LIN {X 0,Y 362.111,Z 381.376,A -85,B 0,C 180,E1 -12954.431,E2 -12954.431} C_VEL
LIN {X 0,Y 362.275,Z 381.356,A -85,B 0,C 180,E1 -12957.776,E2 -12957.776} C_VEL
LIN {X 0,Y 362.422,Z 381.337,A -85,B 0,C 180,E1 -12960,E2 -12960} C_VEL
LIN {X 0,Y 362.276,Z 381.354,A -85,B 0,C 180,E1 -12962.224,E2 -12962.224} C_VEL
LIN {X 0,Y 362.165,Z 381.372,A -85,B 0,C 180,E1 -12966.686,E2 -12966.686} C_VEL
LIN {X 0,Y 362.068,Z 381.386,A -85,B 0,C 180,E1 -12968.933,E2 -12968.933} C_VEL
LIN {X 0,Y 361.959,Z 381.395,A -85,B 0,C 180,E1 -12972.332,E2 -12972.332} C_VEL
LIN {X 0,Y 361.955,Z 381.398,A -85,B 0,C 180,E1 -12974.621,E2 -12974.621} C_VEL
LIN {X 0,Y 361.949,Z 381.396,A -85,B 0,C 180,E1 -12978.1,E2 -12978.1} C_VEL
LIN {X 0,Y 361.885,Z 381.404,A -85,B 0,C 180,E1 -12981.653,E2 -12981.653} C_VEL
LIN {X 0,Y 361.922,Z 381.4,A -85,B 0,C 180,E1 -12985.291,E2 -12985.291} C_VEL
LIN {X 0,Y 361.912,Z 381.4,A -85,B 0,C 180,E1 -12987.779,E2 -12987.779} C_VEL
LIN {X 0,Y 361.841,Z 381.41,A -85,B 0,C 180,E1 -12991.286,E2 -12991.286} C_VEL
LIN {X 0,Y 361.849,Z 381.411,A -85,B 0,C 180,E1 -12994.281,E2 -12994.281} C_VEL
LIN {X 0,Y 361.861,Z 381.407,A -85,B 0,C 180,E1 -12997.224,E2 -12997.224} C_VEL
LIN {X 0,Y 361.901,Z 381.405,A -85,B 0,C 180,E1 -13000.769,E2 -13000.769} C_VEL
LIN {X 0,Y 361.907,Z 381.406,A -85,B 0,C 180,E1 -13004.355,E2 -13004.355} C_VEL
LIN {X 0,Y 361.838,Z 381.41,A -85,B 0,C 180,E1 -13007.568,E2 -13007.568} C_VEL
LIN {X 0,Y 361.87,Z 381.407,A -85,B 0,C 180,E1 -13010.974,E2 -13010.974} C_VEL
LIN {X 0,Y 361.873,Z 381.408,A -85,B 0,C 180,E1 -13014.656,E2 -13014.656} C_VEL
LIN {X 0,Y 361.837,Z 381.416,A -85,B 0,C 180,E1 -13018.371,E2 -13018.371} C_VEL
LIN {X 0,Y 361.92,Z 381.554,A -85,B 0,C 180,E1 -13019.486,E2 -13019.486} C_VEL
LIN {X 0,Y 364.634,Z 393.775,A -85,B 0,C 180,E1 -13022.697,E2 -13022.697} C_VEL
LIN {X 0,Y 366.023,Z 401.747,A -85,B 0,C 180,E1 -13024.694,E2 -13024.694} C_VEL
LIN {X 0,Y 364.596,Z 415.783,A -85,B 0,C 180,E1 -13027.91,E2 -13027.91} C_VEL
LIN {X 0,Y 369.128,Z 442.935,A -85,B 0,C 180,E1 -13028.748,E2 -13028.748} C_VEL
LIN {X 0,Y 370.192,Z 451.075,A -85,B 0,C 180,E1 -13028.977,E2 -13028.977} C_VEL
LIN {X 0,Y 368.952,Z 524.302,A -85,B 0,C 180,E1 -13030.42,E2 -13030.42} C_VEL
LIN {X 0,Y 368.284,Z 537.515,A -85,B 0,C 180,E1 -13030.89,E2 -13030.89} C_VEL
LIN {X 0,Y 367.403,Z 549.648,A -85,B 0,C 180,E1 -13031.53,E2 -13031.53} C_VEL
LIN {X 0,Y 366.36,Z 561.898,A -85,B 0,C 180,E1 -13032.414,E2 -13032.414} C_VEL
LIN {X 0,Y 365.162,Z 573.49,A -85,B 0,C 180,E1 -13033.508,E2 -13033.508} C_VEL
LIN {X 0,Y 364.028,Z 584.075,A -85,B 0,C 180,E1 -13034.768,E2 -13034.768} C_VEL
LIN {X 0,Y 363.201,Z 592.48,A -85,B 0,C 180,E1 -13036.003,E2 -13036.003} C_VEL
LIN {X 0,Y 362.381,Z 600.367,A -85,B 0,C 180,E1 -13037.398,E2 -13037.398} C_VEL
LIN {X 0,Y 361.507,Z 608.07,A -85,B 0,C 180,E1 -13039.074,E2 -13039.074} C_VEL
LIN {X 0,Y 360.907,Z 615.183,A -85,B 0,C 180,E1 -13041.038,E2 -13041.038} C_VEL
LIN {X 0,Y 360.587,Z 619.917,A -85,B 0,C 180,E1 -13042.722,E2 -13042.722} C_VEL
LIN {X 0,Y 360.383,Z 623.535,A -85,B 0,C 180,E1 -13044.404,E2 -13044.404} C_VEL
LIN {X 0,Y 360.365,Z 625.404,A -85,B 0,C 180,E1 -13045.526,E2 -13045.526} C_VEL
LIN {X 0,Y 360.303,Z 626.804,A -85,B 0,C 180,E1 -13046.645,E2 -13046.645} C_VEL
LIN {X 0,Y 360.385,Z 628.417,A -85,B 0,C 180,E1 -13048.883,E2 -13048.883} C_VEL
LIN {X 0,Y 360.424,Z 628.634,A -85,B 0,C 180,E1 -13050,E2 -13050} C_VEL
LIN {X 0,Y 360.385,Z 628.413,A -85,B 0,C 180,E1 -13051.117,E2 -13051.117} C_VEL
LIN {X 0,Y 360.304,Z 626.796,A -85,B 0,C 180,E1 -13053.355,E2 -13053.355} C_VEL
LIN {X 0,Y 360.366,Z 625.392,A -85,B 0,C 180,E1 -13054.474,E2 -13054.474} C_VEL
LIN {X 0,Y 360.378,Z 622.815,A -85,B 0,C 180,E1 -13055.961,E2 -13055.961} C_VEL
LIN {X 0,Y 360.66,Z 618.449,A -85,B 0,C 180,E1 -13057.84,E2 -13057.84} C_VEL
LIN {X 0,Y 361.127,Z 612.315,A -85,B 0,C 180,E1 -13059.804,E2 -13059.804} C_VEL
LIN {X 0,Y 361.753,Z 605.619,A -85,B 0,C 180,E1 -13061.486,E2 -13061.486} C_VEL
LIN {X 0,Y 362.739,Z 597.321,A -85,B 0,C 180,E1 -13063.159,E2 -13063.159} C_VEL
LIN {X 0,Y 363.749,Z 587.774,A -85,B 0,C 180,E1 -13064.699,E2 -13064.699} C_VEL
LIN {X 0,Y 364.751,Z 577.122,A -85,B 0,C 180,E1 -13066.079,E2 -13066.079} C_VEL
LIN {X 0,Y 365.892,Z 566.481,A -85,B 0,C 180,E1 -13067.176,E2 -13067.176} C_VEL
LIN {X 0,Y 366.968,Z 554.588,A -85,B 0,C 180,E1 -13068.132,E2 -13068.132} C_VEL
LIN {X 0,Y 367.917,Z 542.215,A -85,B 0,C 180,E1 -13068.877,E2 -13068.877} C_VEL
LIN {X 0,Y 368.713,Z 529.503,A -85,B 0,C 180,E1 -13069.412,E2 -13069.412} C_VEL
LIN {X 0,Y 369.102,Z 516.14,A -85,B 0,C 180,E1 -13069.753,E2 -13069.753} C_VEL
LIN {X 0,Y 370.066,Z 449.66,A -85,B 0,C 180,E1 -13071.046,E2 -13071.046} C_VEL
LIN {X 0,Y 365.283,Z 419.717,A -85,B 0,C 180,E1 -13071.95,E2 -13071.95} C_VEL
LIN {X 0,Y 364.608,Z 415.73,A -85,B 0,C 180,E1 -13072.09,E2 -13072.09} C_VEL
LIN {X 0,Y 366.013,Z 401.695,A -85,B 0,C 180,E1 -13075.303,E2 -13075.303} C_VEL
LIN {X 0,Y 363.854,Z 390.071,A -85,B 0,C 180,E1 -13078.243,E2 -13078.243} C_VEL
LIN {X 0,Y 361.9,Z 381.408,A -85,B 0,C 180,E1 -13080.554,E2 -13080.554} C_VEL
LIN {X 0,Y 361.853,Z 381.409,A -85,B 0,C 180,E1 -13084.28,E2 -13084.28} C_VEL
LIN {X 0,Y 361.869,Z 381.408,A -85,B 0,C 180,E1 -13087.224,E2 -13087.224} C_VEL
LIN {X 0,Y 361.852,Z 381.408,A -85,B 0,C 180,E1 -13090.758,E2 -13090.758} C_VEL
LIN {X 0,Y 361.844,Z 381.409,A -85,B 0,C 180,E1 -13094.363,E2 -13094.363} C_VEL
LIN {X 0,Y 361.88,Z 381.41,A -85,B 0,C 180,E1 -13097.559,E2 -13097.559} C_VEL
LIN {X 0,Y 361.871,Z 381.407,A -85,B 0,C 180,E1 -13100.972,E2 -13100.972} C_VEL
LIN {X 0,Y 361.869,Z 381.406,A -85,B 0,C 180,E1 -13104.654,E2 -13104.654} C_VEL
LIN {X 0,Y 361.832,Z 381.41,A -85,B 0,C 180,E1 -13108.37,E2 -13108.37} C_VEL
LIN {X 0,Y 361.896,Z 381.405,A -85,B 0,C 180,E1 -13110.955,E2 -13110.955} C_VEL
LIN {X 0,Y 361.948,Z 381.4,A -85,B 0,C 180,E1 -13113.475,E2 -13113.475} C_VEL
LIN {X 0,Y 361.884,Z 381.409,A -85,B 0,C 180,E1 -13117.144,E2 -13117.144} C_VEL
LIN {X 0,Y 361.899,Z 381.403,A -85,B 0,C 180,E1 -13120.723,E2 -13120.723} C_VEL
LIN {X 0,Y 361.926,Z 381.403,A -85,B 0,C 180,E1 -13123.066,E2 -13123.066} C_VEL
LIN {X 0,Y 361.993,Z 381.391,A -85,B 0,C 180,E1 -13126.528,E2 -13126.528} C_VEL
LIN {X 0,Y 362.029,Z 381.385,A -85,B 0,C 180,E1 -13129.938,E2 -13129.938} C_VEL
LIN {X 0,Y 362.143,Z 381.371,A -85,B 0,C 180,E1 -13132.192,E2 -13132.192} C_VEL
LIN {X 0,Y 362.111,Z 381.376,A -85,B 0,C 180,E1 -13134.431,E2 -13134.431} C_VEL
LIN {X 0,Y 362.276,Z 381.355,A -85,B 0,C 180,E1 -13137.776,E2 -13137.776} C_VEL
LIN {X 0,Y 362.422,Z 381.337,A -85,B 0,C 180,E1 -13140,E2 -13140} C_VEL
LIN {X 0,Y 362.276,Z 381.355,A -85,B 0,C 180,E1 -13142.224,E2 -13142.224} C_VEL
LIN {X 0,Y 362.165,Z 381.373,A -85,B 0,C 180,E1 -13146.686,E2 -13146.686} C_VEL
LIN {X 0,Y 362.068,Z 381.386,A -85,B 0,C 180,E1 -13148.933,E2 -13148.933} C_VEL
LIN {X 0,Y 361.959,Z 381.396,A -85,B 0,C 180,E1 -13152.332,E2 -13152.332} C_VEL
LIN {X 0,Y 361.955,Z 381.4,A -85,B 0,C 180,E1 -13154.621,E2 -13154.621} C_VEL
LIN {X 0,Y 361.953,Z 381.396,A -85,B 0,C 180,E1 -13158.1,E2 -13158.1} C_VEL
LIN {X 0,Y 361.886,Z 381.403,A -85,B 0,C 180,E1 -13161.653,E2 -13161.653} C_VEL
LIN {X 0,Y 361.922,Z 381.399,A -85,B 0,C 180,E1 -13165.291,E2 -13165.291} C_VEL
LIN {X 0,Y 361.912,Z 381.4,A -85,B 0,C 180,E1 -13167.779,E2 -13167.779} C_VEL
LIN {X 0,Y 361.841,Z 381.409,A -85,B 0,C 180,E1 -13171.286,E2 -13171.286} C_VEL
LIN {X 0,Y 361.849,Z 381.412,A -85,B 0,C 180,E1 -13174.281,E2 -13174.281} C_VEL
LIN {X 0,Y 361.861,Z 381.407,A -85,B 0,C 180,E1 -13177.224,E2 -13177.224} C_VEL
LIN {X 0,Y 361.902,Z 381.404,A -85,B 0,C 180,E1 -13180.769,E2 -13180.769} C_VEL
LIN {X 0,Y 361.9,Z 381.408,A -85,B 0,C 180,E1 -13184.356,E2 -13184.356} C_VEL
LIN {X 0,Y 361.835,Z 381.41,A -85,B 0,C 180,E1 -13187.569,E2 -13187.569} C_VEL
LIN {X 0,Y 361.87,Z 381.406,A -85,B 0,C 180,E1 -13191.577,E2 -13191.577} C_VEL
LIN {X 0,Y 361.873,Z 381.407,A -85,B 0,C 180,E1 -13194.656,E2 -13194.656} C_VEL
LIN {X 0,Y 361.837,Z 381.414,A -85,B 0,C 180,E1 -13198.371,E2 -13198.371} C_VEL
LIN {X 0,Y 361.909,Z 381.405,A -85,B 0,C 180,E1 -13202.222,E2 -13202.222} C_VEL
LIN {X 0,Y 361.931,Z 381.511,A -85,B 0,C 180,E1 -13205,E2 -13205} C_VEL
LIN {X 0,Y 363.858,Z 391.181,A -85,B 0,C 180,E1 -13207.922,E2 -13207.922} C_VEL
LIN {X 0,Y 367.858,Z 402.665,A -85,B 0,C 180,E1 -13208.433,E2 -13208.433} C_VEL
LIN {X 0,Y 370.625,Z 416.292,A -85,B 0,C 180,E1 -13208.883,E2 -13208.883} C_VEL
LIN {X 0,Y 369.277,Z 498.572,A -85,B 0,C 180,E1 -13210.51,E2 -13210.51} C_VEL
LIN {X 0,Y 368.645,Z 512.357,A -85,B 0,C 180,E1 -13211.018,E2 -13211.018} C_VEL
LIN {X 0,Y 367.922,Z 524.708,A -85,B 0,C 180,E1 -13211.701,E2 -13211.701} C_VEL
LIN {X 0,Y 367.034,Z 536.529,A -85,B 0,C 180,E1 -13212.592,E2 -13212.592} C_VEL
LIN {X 0,Y 366.058,Z 547.685,A -85,B 0,C 180,E1 -13213.673,E2 -13213.673} C_VEL
LIN {X 0,Y 365.101,Z 558.085,A -85,B 0,C 180,E1 -13214.938,E2 -13214.938} C_VEL
LIN {X 0,Y 364.055,Z 567.253,A -85,B 0,C 180,E1 -13216.321,E2 -13216.321} C_VEL
LIN {X 0,Y 362.98,Z 576.155,A -85,B 0,C 180,E1 -13217.987,E2 -13217.987} C_VEL
LIN {X 0,Y 362.153,Z 583.316,A -85,B 0,C 180,E1 -13219.659,E2 -13219.659} C_VEL
LIN {X 0,Y 361.582,Z 588.146,A -85,B 0,C 180,E1 -13221.055,E2 -13221.055} C_VEL
LIN {X 0,Y 361.087,Z 592.838,A -85,B 0,C 180,E1 -13222.733,E2 -13222.733} C_VEL
LIN {X 0,Y 360.833,Z 596.422,A -85,B 0,C 180,E1 -13224.411,E2 -13224.411} C_VEL
LIN {X 0,Y 360.604,Z 598.279,A -85,B 0,C 180,E1 -13225.529,E2 -13225.529} C_VEL
LIN {X 0,Y 360.497,Z 599.674,A -85,B 0,C 180,E1 -13226.647,E2 -13226.647} C_VEL
LIN {X 0,Y 360.421,Z 601.275,A -85,B 0,C 180,E1 -13228.883,E2 -13228.883} C_VEL
LIN {X 0,Y 360.426,Z 601.507,A -85,B 0,C 180,E1 -13230,E2 -13230} C_VEL
LIN {X 0,Y 360.421,Z 601.318,A -85,B 0,C 180,E1 -13231.117,E2 -13231.117} C_VEL
LIN {X 0,Y 360.456,Z 600.735,A -85,B 0,C 180,E1 -13232.235,E2 -13232.235} C_VEL
LIN {X 0,Y 360.602,Z 598.419,A -85,B 0,C 180,E1 -13234.471,E2 -13234.471} C_VEL
LIN {X 0,Y 360.93,Z 595.557,A -85,B 0,C 180,E1 -13236.148,E2 -13236.148} C_VEL
LIN {X 0,Y 361.226,Z 591.682,A -85,B 0,C 180,E1 -13237.827,E2 -13237.827} C_VEL
LIN {X 0,Y 361.741,Z 586.677,A -85,B 0,C 180,E1 -13239.505,E2 -13239.505} C_VEL
LIN {X 0,Y 362.473,Z 580.373,A -85,B 0,C 180,E1 -13241.18,E2 -13241.18} C_VEL
LIN {X 0,Y 363.389,Z 572.48,A -85,B 0,C 180,E1 -13242.85,E2 -13242.85} C_VEL
LIN {X 0,Y 364.398,Z 564.427,A -85,B 0,C 180,E1 -13244.235,E2 -13244.235} C_VEL
LIN {X 0,Y 365.437,Z 554.603,A -85,B 0,C 180,E1 -13245.619,E2 -13245.619} C_VEL
LIN {X 0,Y 366.306,Z 544.935,A -85,B 0,C 180,E1 -13246.725,E2 -13246.725} C_VEL
LIN {X 0,Y 367.254,Z 534.463,A -85,B 0,C 180,E1 -13247.685,E2 -13247.685} C_VEL
LIN {X 0,Y 368.214,Z 521.847,A -85,B 0,C 180,E1 -13248.572,E2 -13248.572} C_VEL
LIN {X 0,Y 368.838,Z 509.216,A -85,B 0,C 180,E1 -13249.225,E2 -13249.225} C_VEL
LIN {X 0,Y 369.326,Z 497.213,A -85,B 0,C 180,E1 -13249.632,E2 -13249.632} C_VEL
LIN {X 0,Y 369.596,Z 480.297,A -85,B 0,C 180,E1 -13249.98,E2 -13249.98} C_VEL
LIN {X 0,Y 369.082,Z 474.486,A -85,B 0,C 180,E1 -13250.127,E2 -13250.127} C_VEL
LIN {X 0,Y 364.083,Z 455.777,A -85,B 0,C 180,E1 -13250.807,E2 -13250.807} C_VEL
LIN {X 0,Y 363.551,Z 449.967,A -85,B 0,C 180,E1 -13250.959,E2 -13250.959} C_VEL
LIN {X 0,Y 363.969,Z 416.729,A -85,B 0,C 180,E1 -13251.624,E2 -13251.624} C_VEL
LIN {X 0,Y 360.737,Z 402.305,A -85,B 0,C 180,E1 -13252.134,E2 -13252.134} C_VEL
LIN {X 0,Y 356.684,Z 391.491,A -85,B 0,C 180,E1 -13252.648,E2 -13252.648} C_VEL
LIN {X 0,Y 354.901,Z 382.279,A -85,B 0,C 180,E1 -13255.512,E2 -13255.512} C_VEL
LIN {X 0,Y 354.846,Z 382.283,A -85,B 0,C 180,E1 -13258.381,E2 -13258.381} C_VEL
LIN {X 0,Y 354.787,Z 382.29,A -85,B 0,C 180,E1 -13262.333,E2 -13262.333} C_VEL
LIN {X 0,Y 354.821,Z 382.288,A -85,B 0,C 180,E1 -13265.699,E2 -13265.699} C_VEL
LIN {X 0,Y 354.822,Z 382.286,A -85,B 0,C 180,E1 -13269.423,E2 -13269.423} C_VEL
LIN {X 0,Y 354.788,Z 382.287,A -85,B 0,C 180,E1 -13272.867,E2 -13272.867} C_VEL
LIN {X 0,Y 354.837,Z 382.283,A -85,B 0,C 180,E1 -13276.114,E2 -13276.114} C_VEL
LIN {X 0,Y 354.854,Z 382.28,A -85,B 0,C 180,E1 -13279.188,E2 -13279.188} C_VEL
LIN {X 0,Y 354.805,Z 382.285,A -85,B 0,C 180,E1 -13282.401,E2 -13282.401} C_VEL
LIN {X 0,Y 354.808,Z 382.286,A -85,B 0,C 180,E1 -13284.94,E2 -13284.94} C_VEL
LIN {X 0,Y 354.789,Z 382.288,A -85,B 0,C 180,E1 -13288.404,E2 -13288.404} C_VEL
LIN {X 0,Y 354.845,Z 382.285,A -85,B 0,C 180,E1 -13291.618,E2 -13291.618} C_VEL
LIN {X 0,Y 354.893,Z 382.275,A -85,B 0,C 180,E1 -13294.172,E2 -13294.172} C_VEL
LIN {X 0,Y 354.829,Z 382.284,A -85,B 0,C 180,E1 -13297.893,E2 -13297.893} C_VEL
LIN {X 0,Y 354.916,Z 382.272,A -85,B 0,C 180,E1 -13301.891,E2 -13301.891} C_VEL
LIN {X 0,Y 354.936,Z 382.27,A -85,B 0,C 180,E1 -13305.981,E2 -13305.981} C_VEL
LIN {X 0,Y 354.975,Z 382.266,A -85,B 0,C 180,E1 -13309.736,E2 -13309.736} C_VEL
LIN {X 0,Y 355.106,Z 382.248,A -85,B 0,C 180,E1 -13312.037,E2 -13312.037} C_VEL
LIN {X 0,Y 355.085,Z 382.25,A -85,B 0,C 180,E1 -13314.321,E2 -13314.321} C_VEL
LIN {X 0,Y 355.239,Z 382.233,A -85,B 0,C 180,E1 -13317.732,E2 -13317.732} C_VEL
LIN {X 0,Y 355.391,Z 382.212,A -85,B 0,C 180,E1 -13320,E2 -13320} C_VEL
LIN {X 0,Y 355.239,Z 382.231,A -85,B 0,C 180,E1 -13322.268,E2 -13322.268} C_VEL
LIN {X 0,Y 355.131,Z 382.249,A -85,B 0,C 180,E1 -13326.819,E2 -13326.819} C_VEL
LIN {X 0,Y 355.01,Z 382.265,A -85,B 0,C 180,E1 -13329.112,E2 -13329.112} C_VEL
LIN {X 0,Y 354.919,Z 382.274,A -85,B 0,C 180,E1 -13332.581,E2 -13332.581} C_VEL
LIN {X 0,Y 354.882,Z 382.276,A -85,B 0,C 180,E1 -13336.096,E2 -13336.096} C_VEL
LIN {X 0,Y 354.894,Z 382.277,A -85,B 0,C 180,E1 -13338.473,E2 -13338.473} C_VEL
LIN {X 0,Y 354.828,Z 382.283,A -85,B 0,C 180,E1 -13342.106,E2 -13342.106} C_VEL
LIN {X 0,Y 354.893,Z 382.274,A -85,B 0,C 180,E1 -13345.828,E2 -13345.828} C_VEL
LIN {X 0,Y 354.848,Z 382.28,A -85,B 0,C 180,E1 -13349.679,E2 -13349.679} C_VEL
LIN {X 0,Y 354.801,Z 382.285,A -85,B 0,C 180,E1 -13353.703,E2 -13353.703} C_VEL
LIN {X 0,Y 354.795,Z 382.292,A -85,B 0,C 180,E1 -13356.46,E2 -13356.46} C_VEL
LIN {X 0,Y 354.82,Z 382.283,A -85,B 0,C 180,E1 -13359.424,E2 -13359.424} C_VEL
LIN {X 0,Y 354.831,Z 382.284,A -85,B 0,C 180,E1 -13362.876,E2 -13362.876} C_VEL
LIN {X 0,Y 354.782,Z 382.291,A -85,B 0,C 180,E1 -13366.107,E2 -13366.107} C_VEL
LIN {X 0,Y 354.804,Z 382.286,A -85,B 0,C 180,E1 -13369.182,E2 -13369.182} C_VEL
LIN {X 0,Y 354.81,Z 382.291,A -85,B 0,C 180,E1 -13372.402,E2 -13372.402} C_VEL
LIN {X 0,Y 354.811,Z 382.287,A -85,B 0,C 180,E1 -13374.942,E2 -13374.942} C_VEL
LIN {X 0,Y 354.793,Z 382.293,A -85,B 0,C 180,E1 -13378.406,E2 -13378.406} C_VEL
LIN {X 0,Y 354.853,Z 382.427,A -85,B 0,C 180,E1 -13379.098,E2 -13379.098} C_VEL
LIN {X 0,Y 357.443,Z 394.03,A -85,B 0,C 180,E1 -13382.225,E2 -13382.225} C_VEL
LIN {X 0,Y 359.044,Z 402.833,A -85,B 0,C 180,E1 -13384.493,E2 -13384.493} C_VEL
LIN {X 0,Y 358.039,Z 413.027,A -85,B 0,C 180,E1 -13386.885,E2 -13386.885} C_VEL
LIN {X 0,Y 357.806,Z 415.48,A -85,B 0,C 180,E1 -13387.461,E2 -13387.461} C_VEL
LIN {X 0,Y 362.538,Z 444.097,A -85,B 0,C 180,E1 -13388.372,E2 -13388.372} C_VEL
LIN {X 0,Y 363.531,Z 452.054,A -85,B 0,C 180,E1 -13388.598,E2 -13388.598} C_VEL
LIN {X 0,Y 362.278,Z 524.048,A -85,B 0,C 180,E1 -13390.044,E2 -13390.044} C_VEL
LIN {X 0,Y 361.562,Z 537.255,A -85,B 0,C 180,E1 -13390.52,E2 -13390.52} C_VEL
LIN {X 0,Y 360.675,Z 549.387,A -85,B 0,C 180,E1 -13391.172,E2 -13391.172} C_VEL
LIN {X 0,Y 359.587,Z 561.635,A -85,B 0,C 180,E1 -13392.072,E2 -13392.072} C_VEL
LIN {X 0,Y 358.324,Z 573.226,A -85,B 0,C 180,E1 -13393.184,E2 -13393.184} C_VEL
LIN {X 0,Y 357.192,Z 583.576,A -85,B 0,C 180,E1 -13394.438,E2 -13394.438} C_VEL
LIN {X 0,Y 356.282,Z 592.214,A -85,B 0,C 180,E1 -13395.725,E2 -13395.725} C_VEL
LIN {X 0,Y 355.422,Z 600.101,A -85,B 0,C 180,E1 -13397.147,E2 -13397.147} C_VEL
LIN {X 0,Y 354.482,Z 607.802,A -85,B 0,C 180,E1 -13398.855,E2 -13398.855} C_VEL
LIN {X 0,Y 353.862,Z 614.915,A -85,B 0,C 180,E1 -13400.858,E2 -13400.858} C_VEL
LIN {X 0,Y 353.51,Z 619.649,A -85,B 0,C 180,E1 -13402.575,E2 -13402.575} C_VEL
LIN {X 0,Y 353.31,Z 623.269,A -85,B 0,C 180,E1 -13404.292,E2 -13404.292} C_VEL
LIN {X 0,Y 353.278,Z 625.137,A -85,B 0,C 180,E1 -13405.436,E2 -13405.436} C_VEL
LIN {X 0,Y 353.225,Z 626.537,A -85,B 0,C 180,E1 -13406.578,E2 -13406.578} C_VEL
LIN {X 0,Y 353.285,Z 628.15,A -85,B 0,C 180,E1 -13408.86,E2 -13408.86} C_VEL
LIN {X 0,Y 353.329,Z 628.367,A -85,B 0,C 180,E1 -13410,E2 -13410} C_VEL
LIN {X 0,Y 353.285,Z 628.146,A -85,B 0,C 180,E1 -13411.14,E2 -13411.14} C_VEL
LIN {X 0,Y 353.225,Z 626.529,A -85,B 0,C 180,E1 -13413.422,E2 -13413.422} C_VEL
LIN {X 0,Y 353.278,Z 625.124,A -85,B 0,C 180,E1 -13414.564,E2 -13414.564} C_VEL
LIN {X 0,Y 353.296,Z 622.818,A -85,B 0,C 180,E1 -13415.937,E2 -13415.937} C_VEL
LIN {X 0,Y 353.605,Z 618.18,A -85,B 0,C 180,E1 -13417.997,E2 -13417.997} C_VEL
LIN {X 0,Y 354.09,Z 612.045,A -85,B 0,C 180,E1 -13420.001,E2 -13420.001} C_VEL
LIN {X 0,Y 354.741,Z 605.348,A -85,B 0,C 180,E1 -13421.716,E2 -13421.716} C_VEL
LIN {X 0,Y 355.797,Z 597.051,A -85,B 0,C 180,E1 -13423.42,E2 -13423.42} C_VEL
LIN {X 0,Y 356.748,Z 588.542,A -85,B 0,C 180,E1 -13424.839,E2 -13424.839} C_VEL
LIN {X 0,Y 357.77,Z 578.028,A -85,B 0,C 180,E1 -13426.255,E2 -13426.255} C_VEL
LIN {X 0,Y 359.104,Z 566.209,A -85,B 0,C 180,E1 -13427.511,E2 -13427.511} C_VEL
LIN {X 0,Y 360.229,Z 554.315,A -85,B 0,C 180,E1 -13428.483,E2 -13428.483} C_VEL
LIN {X 0,Y 361.203,Z 541.941,A -85,B 0,C 180,E1 -13429.241,E2 -13429.241} C_VEL
LIN {X 0,Y 362.017,Z 529.225,A -85,B 0,C 180,E1 -13429.786,E2 -13429.786} C_VEL
LIN {X 0,Y 362.442,Z 515.853,A -85,B 0,C 180,E1 -13430.132,E2 -13430.132} C_VEL
LIN {X 0,Y 363.437,Z 450.516,A -85,B 0,C 180,E1 -13431.425,E2 -13431.425} C_VEL
LIN {X 0,Y 358.744,Z 421.038,A -85,B 0,C 180,E1 -13432.337,E2 -13432.337} C_VEL
LIN {X 0,Y 357.805,Z 415.433,A -85,B 0,C 180,E1 -13432.539,E2 -13432.539} C_VEL
LIN {X 0,Y 359.057,Z 402.761,A -85,B 0,C 180,E1 -13435.506,E2 -13435.506} C_VEL
LIN {X 0,Y 356.836,Z 391.096,A -85,B 0,C 180,E1 -13438.529,E2 -13438.529} C_VEL
LIN {X 0,Y 354.848,Z 382.287,A -85,B 0,C 180,E1 -13440.952,E2 -13440.952} C_VEL
LIN {X 0,Y 354.805,Z 382.292,A -85,B 0,C 180,E1 -13443.701,E2 -13443.701} C_VEL
LIN {X 0,Y 354.799,Z 382.287,A -85,B 0,C 180,E1 -13446.458,E2 -13446.458} C_VEL
LIN {X 0,Y 354.822,Z 382.288,A -85,B 0,C 180,E1 -13449.423,E2 -13449.423} C_VEL
LIN {X 0,Y 354.79,Z 382.288,A -85,B 0,C 180,E1 -13452.867,E2 -13452.867} C_VEL
LIN {X 0,Y 354.848,Z 382.281,A -85,B 0,C 180,E1 -13456.116,E2 -13456.116} C_VEL
LIN {X 0,Y 354.852,Z 382.283,A -85,B 0,C 180,E1 -13459.188,E2 -13459.188} C_VEL
LIN {X 0,Y 354.805,Z 382.285,A -85,B 0,C 180,E1 -13462.401,E2 -13462.401} C_VEL
LIN {X 0,Y 354.807,Z 382.287,A -85,B 0,C 180,E1 -13464.94,E2 -13464.94} C_VEL
LIN {X 0,Y 354.788,Z 382.288,A -85,B 0,C 180,E1 -13468.404,E2 -13468.404} C_VEL
LIN {X 0,Y 354.848,Z 382.283,A -85,B 0,C 180,E1 -13471.619,E2 -13471.619} C_VEL
LIN {X 0,Y 354.893,Z 382.274,A -85,B 0,C 180,E1 -13474.172,E2 -13474.172} C_VEL
LIN {X 0,Y 354.828,Z 382.283,A -85,B 0,C 180,E1 -13477.894,E2 -13477.894} C_VEL
LIN {X 0,Y 354.915,Z 382.272,A -85,B 0,C 180,E1 -13481.891,E2 -13481.891} C_VEL
LIN {X 0,Y 354.936,Z 382.269,A -85,B 0,C 180,E1 -13485.981,E2 -13485.981} C_VEL
LIN {X 0,Y 354.975,Z 382.264,A -85,B 0,C 180,E1 -13489.736,E2 -13489.736} C_VEL
LIN {X 0,Y 355.106,Z 382.248,A -85,B 0,C 180,E1 -13492.037,E2 -13492.037} C_VEL
LIN {X 0,Y 355.085,Z 382.251,A -85,B 0,C 180,E1 -13494.321,E2 -13494.321} C_VEL
LIN {X 0,Y 355.239,Z 382.231,A -85,B 0,C 180,E1 -13497.732,E2 -13497.732} C_VEL
LIN {X 0,Y 355.391,Z 382.212,A -85,B 0,C 180,E1 -13500,E2 -13500} C_VEL
LIN {X 0,Y 355.239,Z 382.232,A -85,B 0,C 180,E1 -13502.268,E2 -13502.268} C_VEL
LIN {X 0,Y 355.131,Z 382.25,A -85,B 0,C 180,E1 -13506.819,E2 -13506.819} C_VEL
LIN {X 0,Y 355.01,Z 382.263,A -85,B 0,C 180,E1 -13509.113,E2 -13509.113} C_VEL
LIN {X 0,Y 354.919,Z 382.275,A -85,B 0,C 180,E1 -13512.581,E2 -13512.581} C_VEL
LIN {X 0,Y 354.883,Z 382.277,A -85,B 0,C 180,E1 -13516.096,E2 -13516.096} C_VEL
LIN {X 0,Y 354.9,Z 382.277,A -85,B 0,C 180,E1 -13518.472,E2 -13518.472} C_VEL
LIN {X 0,Y 354.829,Z 382.284,A -85,B 0,C 180,E1 -13522.107,E2 -13522.107} C_VEL
LIN {X 0,Y 354.893,Z 382.274,A -85,B 0,C 180,E1 -13525.828,E2 -13525.828} C_VEL
LIN {X 0,Y 354.848,Z 382.28,A -85,B 0,C 180,E1 -13529.679,E2 -13529.679} C_VEL
LIN {X 0,Y 354.801,Z 382.286,A -85,B 0,C 180,E1 -13533.703,E2 -13533.703} C_VEL
LIN {X 0,Y 354.795,Z 382.292,A -85,B 0,C 180,E1 -13536.46,E2 -13536.46} C_VEL
LIN {X 0,Y 354.82,Z 382.284,A -85,B 0,C 180,E1 -13539.424,E2 -13539.424} C_VEL
LIN {X 0,Y 354.833,Z 382.284,A -85,B 0,C 180,E1 -13542.876,E2 -13542.876} C_VEL
LIN {X 0,Y 354.781,Z 382.292,A -85,B 0,C 180,E1 -13546.107,E2 -13546.107} C_VEL
LIN {X 0,Y 354.786,Z 382.288,A -85,B 0,C 180,E1 -13549.18,E2 -13549.18} C_VEL
LIN {X 0,Y 354.811,Z 382.289,A -85,B 0,C 180,E1 -13552.402,E2 -13552.402} C_VEL
LIN {X 0,Y 354.811,Z 382.286,A -85,B 0,C 180,E1 -13554.942,E2 -13554.942} C_VEL
LIN {X 0,Y 354.793,Z 382.291,A -85,B 0,C 180,E1 -13558.406,E2 -13558.406} C_VEL
LIN {X 0,Y 354.847,Z 382.282,A -85,B 0,C 180,E1 -13561.619,E2 -13561.619} C_VEL
LIN {X 0,Y 354.894,Z 382.349,A -85,B 0,C 180,E1 -13564.645,E2 -13564.645} C_VEL
LIN {X 0,Y 356.704,Z 391.553,A -85,B 0,C 180,E1 -13567.475,E2 -13567.475} C_VEL
LIN {X 0,Y 361.409,Z 404.429,A -85,B 0,C 180,E1 -13568.059,E2 -13568.059} C_VEL
LIN {X 0,Y 364.059,Z 417.73,A -85,B 0,C 180,E1 -13568.507,E2 -13568.507} C_VEL
LIN {X 0,Y 362.622,Z 498.854,A -85,B 0,C 180,E1 -13570.137,E2 -13570.137} C_VEL
LIN {X 0,Y 362.003,Z 511.874,A -85,B 0,C 180,E1 -13570.619,E2 -13570.619} C_VEL
LIN {X 0,Y 361.211,Z 524.982,A -85,B 0,C 180,E1 -13571.348,E2 -13571.348} C_VEL
LIN {X 0,Y 360.275,Z 536.802,A -85,B 0,C 180,E1 -13572.254,E2 -13572.254} C_VEL
LIN {X 0,Y 359.224,Z 548.27,A -85,B 0,C 180,E1 -13573.389,E2 -13573.389} C_VEL
LIN {X 0,Y 358.272,Z 558.355,A -85,B 0,C 180,E1 -13574.644,E2 -13574.644} C_VEL
LIN {X 0,Y 357.16,Z 567.523,A -85,B 0,C 180,E1 -13576.052,E2 -13576.052} C_VEL
LIN {X 0,Y 356.046,Z 576.424,A -85,B 0,C 180,E1 -13577.749,E2 -13577.749} C_VEL
LIN {X 0,Y 355.186,Z 583.585,A -85,B 0,C 180,E1 -13579.454,E2 -13579.454} C_VEL
LIN {X 0,Y 354.568,Z 588.415,A -85,B 0,C 180,E1 -13580.876,E2 -13580.876} C_VEL
LIN {X 0,Y 354.039,Z 593.106,A -85,B 0,C 180,E1 -13582.587,E2 -13582.587} C_VEL
LIN {X 0,Y 353.769,Z 596.69,A -85,B 0,C 180,E1 -13584.3,E2 -13584.3} C_VEL
LIN {X 0,Y 353.544,Z 598.546,A -85,B 0,C 180,E1 -13585.439,E2 -13585.439} C_VEL
LIN {X 0,Y 353.413,Z 599.942,A -85,B 0,C 180,E1 -13586.58,E2 -13586.58} C_VEL
LIN {X 0,Y 353.327,Z 601.543,A -85,B 0,C 180,E1 -13588.86,E2 -13588.86} C_VEL
LIN {X 0,Y 353.332,Z 601.774,A -85,B 0,C 180,E1 -13590,E2 -13590} C_VEL
LIN {X 0,Y 353.327,Z 601.585,A -85,B 0,C 180,E1 -13591.14,E2 -13591.14} C_VEL
LIN {X 0,Y 353.412,Z 600.039,A -85,B 0,C 180,E1 -13593.42,E2 -13593.42} C_VEL
LIN {X 0,Y 353.542,Z 598.685,A -85,B 0,C 180,E1 -13594.561,E2 -13594.561} C_VEL
LIN {X 0,Y 353.916,Z 595.438,A -85,B 0,C 180,E1 -13596.467,E2 -13596.467} C_VEL
LIN {X 0,Y 354.358,Z 590.394,A -85,B 0,C 180,E1 -13598.554,E2 -13598.554} C_VEL
LIN {X 0,Y 355.157,Z 583.967,A -85,B 0,C 180,E1 -13600.547,E2 -13600.547} C_VEL
LIN {X 0,Y 355.99,Z 576.906,A -85,B 0,C 180,E1 -13602.253,E2 -13602.253} C_VEL
LIN {X 0,Y 357.043,Z 568.103,A -85,B 0,C 180,E1 -13603.953,E2 -13603.953} C_VEL
LIN {X 0,Y 358.17,Z 559.063,A -85,B 0,C 180,E1 -13605.36,E2 -13605.36} C_VEL
LIN {X 0,Y 359.17,Z 548.655,A -85,B 0,C 180,E1 -13606.674,E2 -13606.674} C_VEL
LIN {X 0,Y 360.2,Z 537.918,A -85,B 0,C 180,E1 -13607.75,E2 -13607.75} C_VEL
LIN {X 0,Y 361.224,Z 525.41,A -85,B 0,C 180,E1 -13608.724,E2 -13608.724} C_VEL
LIN {X 0,Y 362.038,Z 512.514,A -85,B 0,C 180,E1 -13609.453,E2 -13609.453} C_VEL
LIN {X 0,Y 362.653,Z 498.66,A -85,B 0,C 180,E1 -13609.972,E2 -13609.972} C_VEL
LIN {X 0,Y 363.551,Z 449.967,A -85,B 0,C 180,E1 -13610.959,E2 -13610.959} C_VEL
LIN {X 0,Y 363.024,Z 444.166,A -85,B 0,C 180,E1 -13611.112,E2 -13611.112} C_VEL
LIN {X 0,Y 358.04,Z 425.501,A -85,B 0,C 180,E1 -13611.82,E2 -13611.82} C_VEL
LIN {X 0,Y 357.478,Z 419.702,A -85,B 0,C 180,E1 -13611.979,E2 -13611.979} C_VEL
LIN {X 0,Y 356.94,Z 415.638,A -85,B 0,C 180,E1 -13612.101,E2 -13612.101} C_VEL
LIN {X 0,Y 354.519,Z 404.948,A -85,B 0,C 180,E1 -13612.492,E2 -13612.492} C_VEL
LIN {X 0,Y 349.547,Z 391.783,A -85,B 0,C 180,E1 -13613.134,E2 -13613.134} C_VEL
LIN {X 0,Y 347.875,Z 383.155,A -85,B 0,C 180,E1 -13615.904,E2 -13615.904} C_VEL
LIN {X 0,Y 347.773,Z 383.166,A -85,B 0,C 180,E1 -13619.66,E2 -13619.66} C_VEL
LIN {X 0,Y 347.741,Z 383.166,A -85,B 0,C 180,E1 -13623.07,E2 -13623.07} C_VEL
LIN {X 0,Y 347.77,Z 383.167,A -85,B 0,C 180,E1 -13626.064,E2 -13626.064} C_VEL
LIN {X 0,Y 347.751,Z 383.165,A -85,B 0,C 180,E1 -13628.792,E2 -13628.792} C_VEL
LIN {X 0,Y 347.749,Z 383.17,A -85,B 0,C 180,E1 -13631.829,E2 -13631.829} C_VEL
LIN {X 0,Y 347.794,Z 383.159,A -85,B 0,C 180,E1 -13635.011,E2 -13635.011} C_VEL
LIN {X 0,Y 347.783,Z 383.16,A -85,B 0,C 180,E1 -13638.39,E2 -13638.39} C_VEL
LIN {X 0,Y 347.772,Z 383.163,A -85,B 0,C 180,E1 -13642.01,E2 -13642.01} C_VEL
LIN {X 0,Y 347.74,Z 383.171,A -85,B 0,C 180,E1 -13645.535,E2 -13645.535} C_VEL
LIN {X 0,Y 347.759,Z 383.168,A -85,B 0,C 180,E1 -13649.653,E2 -13649.653} C_VEL
LIN {X 0,Y 347.846,Z 383.152,A -85,B 0,C 180,E1 -13652.744,E2 -13652.744} C_VEL
LIN {X 0,Y 347.782,Z 383.16,A -85,B 0,C 180,E1 -13656.161,E2 -13656.161} C_VEL
LIN {X 0,Y 347.811,Z 383.158,A -85,B 0,C 180,E1 -13659.909,E2 -13659.909} C_VEL
LIN {X 0,Y 347.86,Z 383.149,A -85,B 0,C 180,E1 -13662.359,E2 -13662.359} C_VEL
LIN {X 0,Y 347.891,Z 383.148,A -85,B 0,C 180,E1 -13665.97,E2 -13665.97} C_VEL
LIN {X 0,Y 347.926,Z 383.145,A -85,B 0,C 180,E1 -13669.525,E2 -13669.525} C_VEL
LIN {X 0,Y 348.066,Z 383.126,A -85,B 0,C 180,E1 -13671.874,E2 -13671.874} C_VEL
LIN {X 0,Y 348.06,Z 383.125,A -85,B 0,C 180,E1 -13674.205,E2 -13674.205} C_VEL
LIN {X 0,Y 348.201,Z 383.109,A -85,B 0,C 180,E1 -13677.686,E2 -13677.686} C_VEL
LIN {X 0,Y 348.361,Z 383.088,A -85,B 0,C 180,E1 -13680,E2 -13680} C_VEL
LIN {X 0,Y 348.201,Z 383.107,A -85,B 0,C 180,E1 -13682.313,E2 -13682.313} C_VEL
LIN {X 0,Y 348.099,Z 383.127,A -85,B 0,C 180,E1 -13686.958,E2 -13686.958} C_VEL
LIN {X 0,Y 347.962,Z 383.14,A -85,B 0,C 180,E1 -13689.299,E2 -13689.299} C_VEL
LIN {X 0,Y 347.886,Z 383.153,A -85,B 0,C 180,E1 -13692.84,E2 -13692.84} C_VEL
LIN {X 0,Y 347.832,Z 383.156,A -85,B 0,C 180,E1 -13696.432,E2 -13696.432} C_VEL
LIN {X 0,Y 347.844,Z 383.157,A -85,B 0,C 180,E1 -13698.861,E2 -13698.861} C_VEL
LIN {X 0,Y 347.768,Z 383.166,A -85,B 0,C 180,E1 -13702.58,E2 -13702.58} C_VEL
LIN {X 0,Y 347.806,Z 383.16,A -85,B 0,C 180,E1 -13705.109,E2 -13705.109} C_VEL
LIN {X 0,Y 347.805,Z 383.158,A -85,B 0,C 180,E1 -13707.694,E2 -13707.694} C_VEL
LIN {X 0,Y 347.758,Z 383.166,A -85,B 0,C 180,E1 -13710.347,E2 -13710.347} C_VEL
LIN {X 0,Y 347.739,Z 383.169,A -85,B 0,C 180,E1 -13714.465,E2 -13714.465} C_VEL
LIN {X 0,Y 347.772,Z 383.162,A -85,B 0,C 180,E1 -13717.99,E2 -13717.99} C_VEL
LIN {X 0,Y 347.78,Z 383.16,A -85,B 0,C 180,E1 -13721.61,E2 -13721.61} C_VEL
LIN {X 0,Y 347.793,Z 383.16,A -85,B 0,C 180,E1 -13725.013,E2 -13725.013} C_VEL
LIN {X 0,Y 347.755,Z 383.169,A -85,B 0,C 180,E1 -13728.397,E2 -13728.397} C_VEL
LIN {X 0,Y 347.775,Z 383.165,A -85,B 0,C 180,E1 -13732.011,E2 -13732.011} C_VEL
LIN {X 0,Y 347.743,Z 383.167,A -85,B 0,C 180,E1 -13735.537,E2 -13735.537} C_VEL
LIN {X 0,Y 347.787,Z 383.255,A -85,B 0,C 180,E1 -13738.687,E2 -13738.687} C_VEL
LIN {X 0,Y 350.429,Z 395.022,A -85,B 0,C 180,E1 -13741.938,E2 -13741.938} C_VEL
LIN {X 0,Y 352.052,Z 403.487,A -85,B 0,C 180,E1 -13744.176,E2 -13744.176} C_VEL
LIN {X 0,Y 351.878,Z 407.69,A -85,B 0,C 180,E1 -13745.202,E2 -13745.202} C_VEL
LIN {X 0,Y 351.019,Z 415.505,A -85,B 0,C 180,E1 -13747.014,E2 -13747.014} C_VEL
LIN {X 0,Y 355.554,Z 442.427,A -85,B 0,C 180,E1 -13747.895,E2 -13747.895} C_VEL
LIN {X 0,Y 356.9,Z 453.026,A -85,B 0,C 180,E1 -13748.206,E2 -13748.206} C_VEL
LIN {X 0,Y 355.63,Z 523.795,A -85,B 0,C 180,E1 -13749.654,E2 -13749.654} C_VEL
LIN {X 0,Y 354.89,Z 536.997,A -85,B 0,C 180,E1 -13750.139,E2 -13750.139} C_VEL
LIN {X 0,Y 353.957,Z 549.126,A -85,B 0,C 180,E1 -13750.801,E2 -13750.801} C_VEL
LIN {X 0,Y 352.835,Z 561.372,A -85,B 0,C 180,E1 -13751.717,E2 -13751.717} C_VEL
LIN {X 0,Y 351.53,Z 572.962,A -85,B 0,C 180,E1 -13752.849,E2 -13752.849} C_VEL
LIN {X 0,Y 350.327,Z 583.368,A -85,B 0,C 180,E1 -13754.133,E2 -13754.133} C_VEL
LIN {X 0,Y 349.381,Z 591.948,A -85,B 0,C 180,E1 -13755.437,E2 -13755.437} C_VEL
LIN {X 0,Y 348.48,Z 599.835,A -85,B 0,C 180,E1 -13756.887,E2 -13756.887} C_VEL
LIN {X 0,Y 347.48,Z 607.535,A -85,B 0,C 180,E1 -13758.627,E2 -13758.627} C_VEL
LIN {X 0,Y 346.804,Z 614.648,A -85,B 0,C 180,E1 -13760.67,E2 -13760.67} C_VEL
LIN {X 0,Y 346.444,Z 619.382,A -85,B 0,C 180,E1 -13762.423,E2 -13762.423} C_VEL
LIN {X 0,Y 346.229,Z 623.002,A -85,B 0,C 180,E1 -13764.175,E2 -13764.175} C_VEL
LIN {X 0,Y 346.176,Z 624.87,A -85,B 0,C 180,E1 -13765.342,E2 -13765.342} C_VEL
LIN {X 0,Y 346.149,Z 626.271,A -85,B 0,C 180,E1 -13766.508,E2 -13766.508} C_VEL
LIN {X 0,Y 346.185,Z 627.883,A -85,B 0,C 180,E1 -13768.837,E2 -13768.837} C_VEL
LIN {X 0,Y 346.234,Z 628.1,A -85,B 0,C 180,E1 -13770,E2 -13770} C_VEL
LIN {X 0,Y 346.185,Z 627.878,A -85,B 0,C 180,E1 -13771.163,E2 -13771.163} C_VEL
LIN {X 0,Y 346.149,Z 626.262,A -85,B 0,C 180,E1 -13773.492,E2 -13773.492} C_VEL
LIN {X 0,Y 346.174,Z 624.855,A -85,B 0,C 180,E1 -13774.658,E2 -13774.658} C_VEL
LIN {X 0,Y 346.245,Z 621.902,A -85,B 0,C 180,E1 -13776.409,E2 -13776.409} C_VEL
LIN {X 0,Y 346.544,Z 617.91,A -85,B 0,C 180,E1 -13778.161,E2 -13778.161} C_VEL
LIN {X 0,Y 347.059,Z 611.775,A -85,B 0,C 180,E1 -13780.206,E2 -13780.206} C_VEL
LIN {X 0,Y 347.758,Z 605.078,A -85,B 0,C 180,E1 -13781.955,E2 -13781.955} C_VEL
LIN {X 0,Y 348.857,Z 596.78,A -85,B 0,C 180,E1 -13783.692,E2 -13783.692} C_VEL
LIN {X 0,Y 349.961,Z 587.115,A -85,B 0,C 180,E1 -13785.31,E2 -13785.31} C_VEL
LIN {X 0,Y 351.089,Z 576.58,A -85,B 0,C 180,E1 -13786.723,E2 -13786.723} C_VEL
LIN {X 0,Y 352.318,Z 565.937,A -85,B 0,C 180,E1 -13787.86,E2 -13787.86} C_VEL
LIN {X 0,Y 353.508,Z 554.042,A -85,B 0,C 180,E1 -13788.848,E2 -13788.848} C_VEL
LIN {X 0,Y 354.51,Z 541.666,A -85,B 0,C 180,E1 -13789.619,E2 -13789.619} C_VEL
LIN {X 0,Y 355.333,Z 528.947,A -85,B 0,C 180,E1 -13790.175,E2 -13790.175} C_VEL
LIN {X 0,Y 355.794,Z 515.566,A -85,B 0,C 180,E1 -13790.524,E2 -13790.524} C_VEL
LIN {X 0,Y 356.775,Z 451.022,A -85,B 0,C 180,E1 -13791.828,E2 -13791.828} C_VEL
LIN {X 0,Y 352.104,Z 421.652,A -85,B 0,C 180,E1 -13792.762,E2 -13792.762} C_VEL
LIN {X 0,Y 351.006,Z 415.118,A -85,B 0,C 180,E1 -13793.012,E2 -13793.012} C_VEL
LIN {X 0,Y 352.113,Z 405.068,A -85,B 0,C 180,E1 -13795.412,E2 -13795.412} C_VEL
LIN {X 0,Y 351.123,Z 398.597,A -85,B 0,C 180,E1 -13797.087,E2 -13797.087} C_VEL
LIN {X 0,Y 348.896,Z 387.914,A -85,B 0,C 180,E1 -13799.983,E2 -13799.983} C_VEL
LIN {X 0,Y 347.77,Z 383.168,A -85,B 0,C 180,E1 -13801.357,E2 -13801.357} C_VEL
LIN {X 0,Y 347.743,Z 383.167,A -85,B 0,C 180,E1 -13804.463,E2 -13804.463} C_VEL
LIN {X 0,Y 347.775,Z 383.164,A -85,B 0,C 180,E1 -13807.989,E2 -13807.989} C_VEL
LIN {X 0,Y 347.754,Z 383.168,A -85,B 0,C 180,E1 -13811.829,E2 -13811.829} C_VEL
LIN {X 0,Y 347.794,Z 383.159,A -85,B 0,C 180,E1 -13815.011,E2 -13815.011} C_VEL
LIN {X 0,Y 347.78,Z 383.161,A -85,B 0,C 180,E1 -13818.39,E2 -13818.39} C_VEL
LIN {X 0,Y 347.772,Z 383.163,A -85,B 0,C 180,E1 -13822.01,E2 -13822.01} C_VEL
LIN {X 0,Y 347.739,Z 383.17,A -85,B 0,C 180,E1 -13825.535,E2 -13825.535} C_VEL
LIN {X 0,Y 347.759,Z 383.166,A -85,B 0,C 180,E1 -13829.653,E2 -13829.653} C_VEL
LIN {X 0,Y 347.847,Z 383.153,A -85,B 0,C 180,E1 -13832.744,E2 -13832.744} C_VEL
LIN {X 0,Y 347.782,Z 383.159,A -85,B 0,C 180,E1 -13836.161,E2 -13836.161} C_VEL
LIN {X 0,Y 347.806,Z 383.158,A -85,B 0,C 180,E1 -13839.909,E2 -13839.909} C_VEL
LIN {X 0,Y 347.859,Z 383.15,A -85,B 0,C 180,E1 -13842.359,E2 -13842.359} C_VEL
LIN {X 0,Y 347.89,Z 383.147,A -85,B 0,C 180,E1 -13845.971,E2 -13845.971} C_VEL
LIN {X 0,Y 347.926,Z 383.143,A -85,B 0,C 180,E1 -13849.526,E2 -13849.526} C_VEL
LIN {X 0,Y 348.066,Z 383.125,A -85,B 0,C 180,E1 -13851.875,E2 -13851.875} C_VEL
LIN {X 0,Y 348.06,Z 383.126,A -85,B 0,C 180,E1 -13854.206,E2 -13854.206} C_VEL
LIN {X 0,Y 348.201,Z 383.107,A -85,B 0,C 180,E1 -13857.687,E2 -13857.687} C_VEL
LIN {X 0,Y 348.361,Z 383.088,A -85,B 0,C 180,E1 -13860,E2 -13860} C_VEL
LIN {X 0,Y 348.201,Z 383.109,A -85,B 0,C 180,E1 -13862.314,E2 -13862.314} C_VEL
LIN {X 0,Y 348.099,Z 383.126,A -85,B 0,C 180,E1 -13866.958,E2 -13866.958} C_VEL
LIN {X 0,Y 347.962,Z 383.139,A -85,B 0,C 180,E1 -13869.299,E2 -13869.299} C_VEL
LIN {X 0,Y 347.886,Z 383.152,A -85,B 0,C 180,E1 -13872.84,E2 -13872.84} C_VEL
LIN {X 0,Y 347.832,Z 383.157,A -85,B 0,C 180,E1 -13876.432,E2 -13876.432} C_VEL
LIN {X 0,Y 347.849,Z 383.155,A -85,B 0,C 180,E1 -13878.861,E2 -13878.861} C_VEL
LIN {X 0,Y 347.768,Z 383.168,A -85,B 0,C 180,E1 -13882.58,E2 -13882.58} C_VEL
LIN {X 0,Y 347.806,Z 383.158,A -85,B 0,C 180,E1 -13885.109,E2 -13885.109} C_VEL
LIN {X 0,Y 347.805,Z 383.157,A -85,B 0,C 180,E1 -13887.695,E2 -13887.695} C_VEL
LIN {X 0,Y 347.758,Z 383.168,A -85,B 0,C 180,E1 -13890.347,E2 -13890.347} C_VEL
LIN {X 0,Y 347.74,Z 383.172,A -85,B 0,C 180,E1 -13894.465,E2 -13894.465} C_VEL
LIN {X 0,Y 347.772,Z 383.163,A -85,B 0,C 180,E1 -13897.99,E2 -13897.99} C_VEL
LIN {X 0,Y 347.782,Z 383.161,A -85,B 0,C 180,E1 -13901.826,E2 -13901.826} C_VEL
LIN {X 0,Y 347.793,Z 383.159,A -85,B 0,C 180,E1 -13905.013,E2 -13905.013} C_VEL
LIN {X 0,Y 347.748,Z 383.17,A -85,B 0,C 180,E1 -13908.398,E2 -13908.398} C_VEL
LIN {X 0,Y 347.775,Z 383.165,A -85,B 0,C 180,E1 -13912.011,E2 -13912.011} C_VEL
LIN {X 0,Y 347.743,Z 383.167,A -85,B 0,C 180,E1 -13915.537,E2 -13915.537} C_VEL
LIN {X 0,Y 347.745,Z 383.17,A -85,B 0,C 180,E1 -13918.301,E2 -13918.301} C_VEL
LIN {X 0,Y 347.778,Z 383.161,A -85,B 0,C 180,E1 -13920.988,E2 -13920.988} C_VEL
LIN {X 0,Y 347.882,Z 383.271,A -85,B 0,C 180,E1 -13924.297,E2 -13924.297} C_VEL
LIN {X 0,Y 349.551,Z 391.914,A -85,B 0,C 180,E1 -13926.989,E2 -13926.989} C_VEL
LIN {X 0,Y 355.129,Z 406.84,A -85,B 0,C 180,E1 -13927.696,E2 -13927.696} C_VEL
LIN {X 0,Y 357.479,Z 419.254,A -85,B 0,C 180,E1 -13928.117,E2 -13928.117} C_VEL
LIN {X 0,Y 355.965,Z 499.137,A -85,B 0,C 180,E1 -13929.75,E2 -13929.75} C_VEL
LIN {X 0,Y 355.331,Z 512.151,A -85,B 0,C 180,E1 -13930.24,E2 -13930.24} C_VEL
LIN {X 0,Y 354.598,Z 524.158,A -85,B 0,C 180,E1 -13930.912,E2 -13930.912} C_VEL
LIN {X 0,Y 353.679,Z 535.49,A -85,B 0,C 180,E1 -13931.762,E2 -13931.762} C_VEL
LIN {X 0,Y 352.618,Z 546.704,A -85,B 0,C 180,E1 -13932.855,E2 -13932.855} C_VEL
LIN {X 0,Y 351.58,Z 557.567,A -85,B 0,C 180,E1 -13934.196,E2 -13934.196} C_VEL
LIN {X 0,Y 350.453,Z 566.104,A -85,B 0,C 180,E1 -13935.483,E2 -13935.483} C_VEL
LIN {X 0,Y 349.48,Z 573.96,A -85,B 0,C 180,E1 -13936.925,E2 -13936.925} C_VEL
LIN {X 0,Y 348.461,Z 581.639,A -85,B 0,C 180,E1 -13938.659,E2 -13938.659} C_VEL
LIN {X 0,Y 347.55,Z 588.684,A -85,B 0,C 180,E1 -13940.69,E2 -13940.69} C_VEL
LIN {X 0,Y 346.987,Z 593.374,A -85,B 0,C 180,E1 -13942.435,E2 -13942.435} C_VEL
LIN {X 0,Y 346.708,Z 596.958,A -85,B 0,C 180,E1 -13944.183,E2 -13944.183} C_VEL
LIN {X 0,Y 346.487,Z 598.813,A -85,B 0,C 180,E1 -13945.346,E2 -13945.346} C_VEL
LIN {X 0,Y 346.333,Z 600.209,A -85,B 0,C 180,E1 -13946.51,E2 -13946.51} C_VEL
LIN {X 0,Y 346.233,Z 601.81,A -85,B 0,C 180,E1 -13948.837,E2 -13948.837} C_VEL
LIN {X 0,Y 346.237,Z 602.041,A -85,B 0,C 180,E1 -13950,E2 -13950} C_VEL
LIN {X 0,Y 346.233,Z 601.852,A -85,B 0,C 180,E1 -13951.163,E2 -13951.163} C_VEL
LIN {X 0,Y 346.332,Z 600.305,A -85,B 0,C 180,E1 -13953.49,E2 -13953.49} C_VEL
LIN {X 0,Y 346.485,Z 598.951,A -85,B 0,C 180,E1 -13954.654,E2 -13954.654} C_VEL
LIN {X 0,Y 346.827,Z 595.946,A -85,B 0,C 180,E1 -13956.478,E2 -13956.478} C_VEL
LIN {X 0,Y 347.141,Z 592.214,A -85,B 0,C 180,E1 -13958.147,E2 -13958.147} C_VEL
LIN {X 0,Y 347.743,Z 587.208,A -85,B 0,C 180,E1 -13959.892,E2 -13959.892} C_VEL
LIN {X 0,Y 348.541,Z 580.904,A -85,B 0,C 180,E1 -13961.633,E2 -13961.633} C_VEL
LIN {X 0,Y 349.546,Z 573.009,A -85,B 0,C 180,E1 -13963.369,E2 -13963.369} C_VEL
LIN {X 0,Y 350.879,Z 563.182,A -85,B 0,C 180,E1 -13965.093,E2 -13965.093} C_VEL
LIN {X 0,Y 351.916,Z 553.667,A -85,B 0,C 180,E1 -13966.432,E2 -13966.432} C_VEL
LIN {X 0,Y 352.981,Z 542.654,A -85,B 0,C 180,E1 -13967.676,E2 -13967.676} C_VEL
LIN {X 0,Y 354.102,Z 531.465,A -85,B 0,C 180,E1 -13968.665,E2 -13968.665} C_VEL
LIN {X 0,Y 354.985,Z 520.107,A -85,B 0,C 180,E1 -13969.442,E2 -13969.442} C_VEL
LIN {X 0,Y 355.663,Z 507.129,A -85,B 0,C 180,E1 -13970.08,E2 -13970.08} C_VEL
LIN {X 0,Y 356.111,Z 493.216,A -85,B 0,C 180,E1 -13970.505,E2 -13970.505} C_VEL
LIN {X 0,Y 357.478,Z 419.702,A -85,B 0,C 180,E1 -13971.979,E2 -13971.979} C_VEL
LIN {X 0,Y 356.958,Z 415.931,A -85,B 0,C 180,E1 -13972.094,E2 -13972.094} C_VEL
LIN {X 0,Y 354.716,Z 410.743,A -85,B 0,C 180,E1 -13972.354,E2 -13972.354} C_VEL
LIN {X 0,Y 351.5,Z 406.106,A -85,B 0,C 180,E1 -13972.673,E2 -13972.673} C_VEL
LIN {X 0,Y 346.648,Z 400.009,A -85,B 0,C 180,E1 -13973.147,E2 -13973.147} C_VEL
LIN {X 0,Y 343.554,Z 395.061,A -85,B 0,C 180,E1 -13973.481,E2 -13973.481} C_VEL
LIN {X 0,Y 342.761,Z 393.258,A -85,B 0,C 180,E1 -13973.58,E2 -13973.58} C_VEL
LIN {X 0,Y 342.376,Z 391.956,A -85,B 0,C 180,E1 -13973.678,E2 -13973.678} C_VEL
LIN {X 0,Y 340.802,Z 384.035,A -85,B 0,C 180,E1 -13976.236,E2 -13976.236} C_VEL
LIN {X 0,Y 340.737,Z 384.044,A -85,B 0,C 180,E1 -13979.97,E2 -13979.97} C_VEL
LIN {X 0,Y 340.693,Z 384.048,A -85,B 0,C 180,E1 -13983.846,E2 -13983.846} C_VEL
LIN {X 0,Y 340.704,Z 384.043,A -85,B 0,C 180,E1 -13986.741,E2 -13986.741} C_VEL
LIN {X 0,Y 340.686,Z 384.047,A -85,B 0,C 180,E1 -13990.246,E2 -13990.246} C_VEL
LIN {X 0,Y 340.674,Z 384.052,A -85,B 0,C 180,E1 -13993.777,E2 -13993.777} C_VEL
LIN {X 0,Y 340.736,Z 384.036,A -85,B 0,C 180,E1 -13997.105,E2 -13997.105} C_VEL
LIN {X 0,Y 340.731,Z 384.04,A -85,B 0,C 180,E1 -14000.252,E2 -14000.252} C_VEL
LIN {X 0,Y 340.707,Z 384.046,A -85,B 0,C 180,E1 -14003.558,E2 -14003.558} C_VEL
LIN {X 0,Y 340.689,Z 384.044,A -85,B 0,C 180,E1 -14006.153,E2 -14006.153} C_VEL
LIN {X 0,Y 340.769,Z 384.034,A -85,B 0,C 180,E1 -14010.332,E2 -14010.332} C_VEL
LIN {X 0,Y 340.799,Z 384.032,A -85,B 0,C 180,E1 -14013.019,E2 -14013.019} C_VEL
LIN {X 0,Y 340.723,Z 384.04,A -85,B 0,C 180,E1 -14016.927,E2 -14016.927} C_VEL
LIN {X 0,Y 340.788,Z 384.032,A -85,B 0,C 180,E1 -14020.733,E2 -14020.733} C_VEL
LIN {X 0,Y 340.78,Z 384.036,A -85,B 0,C 180,E1 -14023.218,E2 -14023.218} C_VEL
LIN {X 0,Y 340.84,Z 384.028,A -85,B 0,C 180,E1 -14026.89,E2 -14026.89} C_VEL
LIN {X 0,Y 340.923,Z 384.015,A -85,B 0,C 180,E1 -14030.507,E2 -14030.507} C_VEL
LIN {X 0,Y 341.068,Z 384,A -85,B 0,C 180,E1 -14032.898,E2 -14032.898} C_VEL
LIN {X 0,Y 341.163,Z 383.987,A -85,B 0,C 180,E1 -14037.639,E2 -14037.639} C_VEL
LIN {X 0,Y 341.31,Z 383.966,A -85,B 0,C 180,E1 -14040,E2 -14040} C_VEL
LIN {X 0,Y 341.163,Z 383.983,A -85,B 0,C 180,E1 -14042.361,E2 -14042.361} C_VEL
LIN {X 0,Y 341.068,Z 384,A -85,B 0,C 180,E1 -14047.102,E2 -14047.102} C_VEL
LIN {X 0,Y 340.868,Z 384.025,A -85,B 0,C 180,E1 -14050.694,E2 -14050.694} C_VEL
LIN {X 0,Y 340.856,Z 384.023,A -85,B 0,C 180,E1 -14054.325,E2 -14054.325} C_VEL
LIN {X 0,Y 340.83,Z 384.029,A -85,B 0,C 180,E1 -14058.467,E2 -14058.467} C_VEL
LIN {X 0,Y 340.748,Z 384.037,A -85,B 0,C 180,E1 -14061.857,E2 -14061.857} C_VEL
LIN {X 0,Y 340.766,Z 384.034,A -85,B 0,C 180,E1 -14065.665,E2 -14065.665} C_VEL
LIN {X 0,Y 340.735,Z 384.041,A -85,B 0,C 180,E1 -14068.32,E2 -14068.32} C_VEL
LIN {X 0,Y 340.698,Z 384.045,A -85,B 0,C 180,E1 -14071.045,E2 -14071.045} C_VEL
LIN {X 0,Y 340.713,Z 384.041,A -85,B 0,C 180,E1 -14075.28,E2 -14075.28} C_VEL
LIN {X 0,Y 340.714,Z 384.044,A -85,B 0,C 180,E1 -14078.389,E2 -14078.389} C_VEL
LIN {X 0,Y 340.721,Z 384.04,A -85,B 0,C 180,E1 -14081.304,E2 -14081.304} C_VEL
LIN {X 0,Y 340.734,Z 384.044,A -85,B 0,C 180,E1 -14084.53,E2 -14084.53} C_VEL
LIN {X 0,Y 340.691,Z 384.048,A -85,B 0,C 180,E1 -14088.692,E2 -14088.692} C_VEL
LIN {X 0,Y 340.734,Z 384.04,A -85,B 0,C 180,E1 -14091.774,E2 -14091.774} C_VEL
LIN {X 0,Y 340.721,Z 384.043,A -85,B 0,C 180,E1 -14095.596,E2 -14095.596} C_VEL
LIN {X 0,Y 340.721,Z 384.123,A -85,B 0,C 180,E1 -14098.266,E2 -14098.266} C_VEL
LIN {X 0,Y 343.086,Z 394.364,A -85,B 0,C 180,E1 -14101.184,E2 -14101.184} C_VEL
LIN {X 0,Y 344.901,Z 403.651,A -85,B 0,C 180,E1 -14103.713,E2 -14103.713} C_VEL
LIN {X 0,Y 345.116,Z 407.424,A -85,B 0,C 180,E1 -14104.682,E2 -14104.682} C_VEL
LIN {X 0,Y 344.196,Z 414.952,A -85,B 0,C 180,E1 -14106.52,E2 -14106.52} C_VEL
LIN {X 0,Y 348.993,Z 443.384,A -85,B 0,C 180,E1 -14107.483,E2 -14107.483} C_VEL
LIN {X 0,Y 350.318,Z 453.371,A -85,B 0,C 180,E1 -14107.788,E2 -14107.788} C_VEL
LIN {X 0,Y 348.969,Z 523.54,A -85,B 0,C 180,E1 -14109.248,E2 -14109.248} C_VEL
LIN {X 0,Y 348.201,Z 536.738,A -85,B 0,C 180,E1 -14109.741,E2 -14109.741} C_VEL
LIN {X 0,Y 347.246,Z 548.865,A -85,B 0,C 180,E1 -14110.415,E2 -14110.415} C_VEL
LIN {X 0,Y 346.097,Z 561.11,A -85,B 0,C 180,E1 -14111.348,E2 -14111.348} C_VEL
LIN {X 0,Y 344.735,Z 572.698,A -85,B 0,C 180,E1 -14112.501,E2 -14112.501} C_VEL
LIN {X 0,Y 343.41,Z 583.46,A -85,B 0,C 180,E1 -14113.855,E2 -14113.855} C_VEL
LIN {X 0,Y 342.262,Z 593.36,A -85,B 0,C 180,E1 -14115.432,E2 -14115.432} C_VEL
LIN {X 0,Y 341.169,Z 602.309,A -85,B 0,C 180,E1 -14117.206,E2 -14117.206} C_VEL
LIN {X 0,Y 340.26,Z 609.512,A -85,B 0,C 180,E1 -14118.986,E2 -14118.986} C_VEL
LIN {X 0,Y 339.61,Z 616.08,A -85,B 0,C 180,E1 -14121.071,E2 -14121.071} C_VEL
LIN {X 0,Y 339.269,Z 620.43,A -85,B 0,C 180,E1 -14122.86,E2 -14122.86} C_VEL
LIN {X 0,Y 339.135,Z 622.838,A -85,B 0,C 180,E1 -14124.11,E2 -14124.11} C_VEL
LIN {X 0,Y 339.079,Z 624.602,A -85,B 0,C 180,E1 -14125.244,E2 -14125.244} C_VEL
LIN {X 0,Y 339.073,Z 626.005,A -85,B 0,C 180,E1 -14126.435,E2 -14126.435} C_VEL
LIN {X 0,Y 339.086,Z 627.616,A -85,B 0,C 180,E1 -14128.812,E2 -14128.812} C_VEL
LIN {X 0,Y 339.139,Z 627.833,A -85,B 0,C 180,E1 -14130,E2 -14130} C_VEL
LIN {X 0,Y 339.086,Z 627.611,A -85,B 0,C 180,E1 -14131.188,E2 -14131.188} C_VEL
LIN {X 0,Y 339.073,Z 625.994,A -85,B 0,C 180,E1 -14133.565,E2 -14133.565} C_VEL
LIN {X 0,Y 339.075,Z 624.587,A -85,B 0,C 180,E1 -14134.756,E2 -14134.756} C_VEL
LIN {X 0,Y 339.168,Z 621.633,A -85,B 0,C 180,E1 -14136.544,E2 -14136.544} C_VEL
LIN {X 0,Y 339.477,Z 617.641,A -85,B 0,C 180,E1 -14138.332,E2 -14138.332} C_VEL
LIN {X 0,Y 340.042,Z 611.505,A -85,B 0,C 180,E1 -14140.419,E2 -14140.419} C_VEL
LIN {X 0,Y 340.794,Z 604.808,A -85,B 0,C 180,E1 -14142.203,E2 -14142.203} C_VEL
LIN {X 0,Y 341.918,Z 596.509,A -85,B 0,C 180,E1 -14143.976,E2 -14143.976} C_VEL
LIN {X 0,Y 342.966,Z 587.999,A -85,B 0,C 180,E1 -14145.449,E2 -14145.449} C_VEL
LIN {X 0,Y 344.116,Z 577.486,A -85,B 0,C 180,E1 -14146.919,E2 -14146.919} C_VEL
LIN {X 0,Y 345.557,Z 565.665,A -85,B 0,C 180,E1 -14148.222,E2 -14148.222} C_VEL
LIN {X 0,Y 346.777,Z 553.769,A -85,B 0,C 180,E1 -14149.228,E2 -14149.228} C_VEL
LIN {X 0,Y 347.839,Z 541.392,A -85,B 0,C 180,E1 -14150.012,E2 -14150.012} C_VEL
LIN {X 0,Y 348.682,Z 528.669,A -85,B 0,C 180,E1 -14150.577,E2 -14150.577} C_VEL
LIN {X 0,Y 349.164,Z 515.279,A -85,B 0,C 180,E1 -14150.932,E2 -14150.932} C_VEL
LIN {X 0,Y 350.205,Z 451.925,A -85,B 0,C 180,E1 -14152.234,E2 -14152.234} C_VEL
LIN {X 0,Y 345.508,Z 422.453,A -85,B 0,C 180,E1 -14153.198,E2 -14153.198} C_VEL
LIN {X 0,Y 344.204,Z 414.879,A -85,B 0,C 180,E1 -14153.484,E2 -14153.484} C_VEL
LIN {X 0,Y 345.116,Z 407.354,A -85,B 0,C 180,E1 -14155.318,E2 -14155.318} C_VEL
LIN {X 0,Y 344.872,Z 403.625,A -85,B 0,C 180,E1 -14156.278,E2 -14156.278} C_VEL
LIN {X 0,Y 342.791,Z 393.053,A -85,B 0,C 180,E1 -14159.16,E2 -14159.16} C_VEL
LIN {X 0,Y 340.721,Z 384.048,A -85,B 0,C 180,E1 -14161.734,E2 -14161.734} C_VEL
LIN {X 0,Y 340.717,Z 384.045,A -85,B 0,C 180,E1 -14165.278,E2 -14165.278} C_VEL
LIN {X 0,Y 340.711,Z 384.042,A -85,B 0,C 180,E1 -14168.386,E2 -14168.386} C_VEL
LIN {X 0,Y 340.701,Z 384.044,A -85,B 0,C 180,E1 -14172.046,E2 -14172.046} C_VEL
LIN {X 0,Y 340.734,Z 384.04,A -85,B 0,C 180,E1 -14175.47,E2 -14175.47} C_VEL
LIN {X 0,Y 340.721,Z 384.04,A -85,B 0,C 180,E1 -14178.696,E2 -14178.696} C_VEL
LIN {X 0,Y 340.735,Z 384.041,A -85,B 0,C 180,E1 -14181.773,E2 -14181.773} C_VEL
LIN {X 0,Y 340.718,Z 384.044,A -85,B 0,C 180,E1 -14185.595,E2 -14185.595} C_VEL
LIN {X 0,Y 340.699,Z 384.045,A -85,B 0,C 180,E1 -14188.955,E2 -14188.955} C_VEL
LIN {X 0,Y 340.774,Z 384.033,A -85,B 0,C 180,E1 -14192.473,E2 -14192.473} C_VEL
LIN {X 0,Y 340.75,Z 384.037,A -85,B 0,C 180,E1 -14195.638,E2 -14195.638} C_VEL
LIN {X 0,Y 340.739,Z 384.041,A -85,B 0,C 180,E1 -14199.474,E2 -14199.474} C_VEL
LIN {X 0,Y 340.851,Z 384.022,A -85,B 0,C 180,E1 -14201.984,E2 -14201.984} C_VEL
LIN {X 0,Y 340.863,Z 384.024,A -85,B 0,C 180,E1 -14205.705,E2 -14205.705} C_VEL
LIN {X 0,Y 340.868,Z 384.023,A -85,B 0,C 180,E1 -14209.306,E2 -14209.306} C_VEL
LIN {X 0,Y 341.068,Z 384.001,A -85,B 0,C 180,E1 -14212.898,E2 -14212.898} C_VEL
LIN {X 0,Y 341.163,Z 383.984,A -85,B 0,C 180,E1 -14217.639,E2 -14217.639} C_VEL
LIN {X 0,Y 341.31,Z 383.967,A -85,B 0,C 180,E1 -14220,E2 -14220} C_VEL
LIN {X 0,Y 341.163,Z 383.986,A -85,B 0,C 180,E1 -14222.361,E2 -14222.361} C_VEL
LIN {X 0,Y 341.068,Z 384,A -85,B 0,C 180,E1 -14227.102,E2 -14227.102} C_VEL
LIN {X 0,Y 340.868,Z 384.027,A -85,B 0,C 180,E1 -14230.694,E2 -14230.694} C_VEL
LIN {X 0,Y 340.856,Z 384.024,A -85,B 0,C 180,E1 -14234.325,E2 -14234.325} C_VEL
LIN {X 0,Y 340.831,Z 384.03,A -85,B 0,C 180,E1 -14238.467,E2 -14238.467} C_VEL
LIN {X 0,Y 340.748,Z 384.037,A -85,B 0,C 180,E1 -14241.857,E2 -14241.857} C_VEL
LIN {X 0,Y 340.767,Z 384.033,A -85,B 0,C 180,E1 -14245.665,E2 -14245.665} C_VEL
LIN {X 0,Y 340.736,Z 384.042,A -85,B 0,C 180,E1 -14248.32,E2 -14248.32} C_VEL
LIN {X 0,Y 340.698,Z 384.043,A -85,B 0,C 180,E1 -14251.045,E2 -14251.045} C_VEL
LIN {X 0,Y 340.714,Z 384.041,A -85,B 0,C 180,E1 -14255.28,E2 -14255.28} C_VEL
LIN {X 0,Y 340.714,Z 384.046,A -85,B 0,C 180,E1 -14258.389,E2 -14258.389} C_VEL
LIN {X 0,Y 340.723,Z 384.039,A -85,B 0,C 180,E1 -14261.304,E2 -14261.304} C_VEL
LIN {X 0,Y 340.733,Z 384.042,A -85,B 0,C 180,E1 -14264.531,E2 -14264.531} C_VEL
LIN {X 0,Y 340.684,Z 384.047,A -85,B 0,C 180,E1 -14268.691,E2 -14268.691} C_VEL
LIN {X 0,Y 340.734,Z 384.04,A -85,B 0,C 180,E1 -14271.774,E2 -14271.774} C_VEL
LIN {X 0,Y 340.722,Z 384.042,A -85,B 0,C 180,E1 -14275.596,E2 -14275.596} C_VEL
LIN {X 0,Y 340.698,Z 384.044,A -85,B 0,C 180,E1 -14278.956,E2 -14278.956} C_VEL
LIN {X 0,Y 340.804,Z 384.029,A -85,B 0,C 180,E1 -14283.021,E2 -14283.021} C_VEL
LIN {X 0,Y 340.829,Z 384.205,A -85,B 0,C 180,E1 -14283.931,E2 -14283.931} C_VEL
LIN {X 0,Y 342.385,Z 392.034,A -85,B 0,C 180,E1 -14286.46,E2 -14286.46} C_VEL
LIN {X 0,Y 348.727,Z 408.695,A -85,B 0,C 180,E1 -14287.299,E2 -14287.299} C_VEL
LIN {X 0,Y 350.828,Z 418.904,A -85,B 0,C 180,E1 -14287.666,E2 -14287.666} C_VEL
LIN {X 0,Y 349.336,Z 499.419,A -85,B 0,C 180,E1 -14289.348,E2 -14289.348} C_VEL
LIN {X 0,Y 348.686,Z 512.428,A -85,B 0,C 180,E1 -14289.847,E2 -14289.847} C_VEL
LIN {X 0,Y 347.927,Z 524.432,A -85,B 0,C 180,E1 -14290.532,E2 -14290.532} C_VEL
LIN {X 0,Y 346.97,Z 535.762,A -85,B 0,C 180,E1 -14291.397,E2 -14291.397} C_VEL
LIN {X 0,Y 345.826,Z 547.116,A -85,B 0,C 180,E1 -14292.524,E2 -14292.524} C_VEL
LIN {X 0,Y 344.76,Z 557.838,A -85,B 0,C 180,E1 -14293.875,E2 -14293.875} C_VEL
LIN {X 0,Y 343.596,Z 566.373,A -85,B 0,C 180,E1 -14295.187,E2 -14295.187} C_VEL
LIN {X 0,Y 342.574,Z 574.23,A -85,B 0,C 180,E1 -14296.656,E2 -14296.656} C_VEL
LIN {X 0,Y 341.504,Z 581.908,A -85,B 0,C 180,E1 -14298.425,E2 -14298.425} C_VEL
LIN {X 0,Y 340.552,Z 588.952,A -85,B 0,C 180,E1 -14300.497,E2 -14300.497} C_VEL
LIN {X 0,Y 339.947,Z 593.642,A -85,B 0,C 180,E1 -14302.277,E2 -14302.277} C_VEL
LIN {X 0,Y 339.649,Z 597.226,A -85,B 0,C 180,E1 -14304.062,E2 -14304.062} C_VEL
LIN {X 0,Y 339.431,Z 599.08,A -85,B 0,C 180,E1 -14305.249,E2 -14305.249} C_VEL
LIN {X 0,Y 339.258,Z 600.476,A -85,B 0,C 180,E1 -14306.437,E2 -14306.437} C_VEL
LIN {X 0,Y 339.139,Z 602.077,A -85,B 0,C 180,E1 -14308.813,E2 -14308.813} C_VEL
LIN {X 0,Y 339.143,Z 602.308,A -85,B 0,C 180,E1 -14310,E2 -14310} C_VEL
LIN {X 0,Y 339.138,Z 602.119,A -85,B 0,C 180,E1 -14311.187,E2 -14311.187} C_VEL
LIN {X 0,Y 339.256,Z 600.571,A -85,B 0,C 180,E1 -14313.563,E2 -14313.563} C_VEL
LIN {X 0,Y 339.429,Z 599.217,A -85,B 0,C 180,E1 -14314.751,E2 -14314.751} C_VEL
LIN {X 0,Y 339.858,Z 595.485,A -85,B 0,C 180,E1 -14316.972,E2 -14316.972} C_VEL
LIN {X 0,Y 340.312,Z 590.926,A -85,B 0,C 180,E1 -14318.91,E2 -14318.91} C_VEL
LIN {X 0,Y 341.209,Z 584.498,A -85,B 0,C 180,E1 -14320.983,E2 -14320.983} C_VEL
LIN {X 0,Y 342.129,Z 577.435,A -85,B 0,C 180,E1 -14322.757,E2 -14322.757} C_VEL
LIN {X 0,Y 343.323,Z 568.63,A -85,B 0,C 180,E1 -14324.522,E2 -14324.522} C_VEL
LIN {X 0,Y 344.517,Z 559.59,A -85,B 0,C 180,E1 -14325.985,E2 -14325.985} C_VEL
LIN {X 0,Y 345.529,Z 549.962,A -85,B 0,C 180,E1 -14327.26,E2 -14327.26} C_VEL
LIN {X 0,Y 346.594,Z 540.016,A -85,B 0,C 180,E1 -14328.318,E2 -14328.318} C_VEL
LIN {X 0,Y 347.706,Z 527.909,A -85,B 0,C 180,E1 -14329.328,E2 -14329.328} C_VEL
LIN {X 0,Y 348.588,Z 515.222,A -85,B 0,C 180,E1 -14330.12,E2 -14330.12} C_VEL
LIN {X 0,Y 349.264,Z 502.577,A -85,B 0,C 180,E1 -14330.656,E2 -14330.656} C_VEL
LIN {X 0,Y 349.591,Z 484.644,A -85,B 0,C 180,E1 -14331.098,E2 -14331.098} C_VEL
LIN {X 0,Y 350.853,Z 419.006,A -85,B 0,C 180,E1 -14332.437,E2 -14332.437} C_VEL
LIN {X 0,Y 348.235,Z 407.346,A -85,B 0,C 180,E1 -14332.873,E2 -14332.873} C_VEL
LIN {X 0,Y 342.761,Z 393.258,A -85,B 0,C 180,E1 -14333.58,E2 -14333.58} C_VEL
LIN {X 0,Y 341.655,Z 391.93,A -85,B 0,C 180,E1 -14333.774,E2 -14333.774} C_VEL
LIN {X 0,Y 337.562,Z 389.718,A -85,B 0,C 180,E1 -14334.774,E2 -14334.774} C_VEL
LIN {X 0,Y 335.105,Z 387.8,A -85,B 0,C 180,E1 -14335.653,E2 -14335.653} C_VEL
LIN {X 0,Y 333.817,Z 385.155,A -85,B 0,C 180,E1 -14336.553,E2 -14336.553} C_VEL
LIN {X 0,Y 333.78,Z 384.906,A -85,B 0,C 180,E1 -14336.916,E2 -14336.916} C_VEL
LIN {X 0,Y 333.69,Z 384.918,A -85,B 0,C 180,E1 -14340.362,E2 -14340.362} C_VEL
LIN {X 0,Y 333.673,Z 384.919,A -85,B 0,C 180,E1 -14344.658,E2 -14344.658} C_VEL
LIN {X 0,Y 333.651,Z 384.925,A -85,B 0,C 180,E1 -14347.65,E2 -14347.65} C_VEL
LIN {X 0,Y 333.645,Z 384.922,A -85,B 0,C 180,E1 -14350.767,E2 -14350.767} C_VEL
LIN {X 0,Y 333.64,Z 384.924,A -85,B 0,C 180,E1 -14354.258,E2 -14354.258} C_VEL
LIN {X 0,Y 333.692,Z 384.916,A -85,B 0,C 180,E1 -14357.626,E2 -14357.626} C_VEL
LIN {X 0,Y 333.679,Z 384.919,A -85,B 0,C 180,E1 -14361.195,E2 -14361.195} C_VEL
LIN {X 0,Y 333.681,Z 384.92,A -85,B 0,C 180,E1 -14365.225,E2 -14365.225} C_VEL
LIN {X 0,Y 333.629,Z 384.924,A -85,B 0,C 180,E1 -14368.222,E2 -14368.222} C_VEL
LIN {X 0,Y 333.705,Z 384.915,A -85,B 0,C 180,E1 -14371.027,E2 -14371.027} C_VEL
LIN {X 0,Y 333.73,Z 384.914,A -85,B 0,C 180,E1 -14373.753,E2 -14373.753} C_VEL
LIN {X 0,Y 333.714,Z 384.914,A -85,B 0,C 180,E1 -14377.913,E2 -14377.913} C_VEL
LIN {X 0,Y 333.788,Z 384.905,A -85,B 0,C 180,E1 -14381.589,E2 -14381.589} C_VEL
LIN {X 0,Y 333.802,Z 384.905,A -85,B 0,C 180,E1 -14385.576,E2 -14385.576} C_VEL
LIN {X 0,Y 333.83,Z 384.901,A -85,B 0,C 180,E1 -14389.078,E2 -14389.078} C_VEL
LIN {X 0,Y 334.018,Z 384.877,A -85,B 0,C 180,E1 -14392.747,E2 -14392.747} C_VEL
LIN {X 0,Y 333.806,Z 384.904,A -85,B 0,C 180,E1 -14395.169,E2 -14395.169} C_VEL
LIN {X 0,Y 334.1,Z 384.867,A -85,B 0,C 180,E1 -14397.589,E2 -14397.589} C_VEL
LIN {X 0,Y 334.26,Z 384.845,A -85,B 0,C 180,E1 -14400,E2 -14400} C_VEL
LIN {X 0,Y 334.101,Z 384.862,A -85,B 0,C 180,E1 -14402.411,E2 -14402.411} C_VEL
LIN {X 0,Y 334.018,Z 384.876,A -85,B 0,C 180,E1 -14407.253,E2 -14407.253} C_VEL
LIN {X 0,Y 333.831,Z 384.903,A -85,B 0,C 180,E1 -14410.922,E2 -14410.922} C_VEL
LIN {X 0,Y 333.802,Z 384.903,A -85,B 0,C 180,E1 -14414.635,E2 -14414.635} C_VEL
LIN {X 0,Y 333.789,Z 384.908,A -85,B 0,C 180,E1 -14418.655,E2 -14418.655} C_VEL
LIN {X 0,Y 333.686,Z 384.918,A -85,B 0,C 180,E1 -14422.279,E2 -14422.279} C_VEL
LIN {X 0,Y 333.73,Z 384.912,A -85,B 0,C 180,E1 -14426.247,E2 -14426.247} C_VEL
LIN {X 0,Y 333.705,Z 384.917,A -85,B 0,C 180,E1 -14428.973,E2 -14428.973} C_VEL
LIN {X 0,Y 333.638,Z 384.927,A -85,B 0,C 180,E1 -14432.587,E2 -14432.587} C_VEL
LIN {X 0,Y 333.672,Z 384.919,A -85,B 0,C 180,E1 -14436.14,E2 -14436.14} C_VEL
LIN {X 0,Y 333.68,Z 384.917,A -85,B 0,C 180,E1 -14439.188,E2 -14439.188} C_VEL
LIN {X 0,Y 333.686,Z 384.921,A -85,B 0,C 180,E1 -14442.512,E2 -14442.512} C_VEL
LIN {X 0,Y 333.632,Z 384.925,A -85,B 0,C 180,E1 -14445.962,E2 -14445.962} C_VEL
LIN {X 0,Y 333.649,Z 384.922,A -85,B 0,C 180,E1 -14449.315,E2 -14449.315} C_VEL
LIN {X 0,Y 333.665,Z 384.921,A -85,B 0,C 180,E1 -14453.168,E2 -14453.168} C_VEL
LIN {X 0,Y 333.637,Z 384.927,A -85,B 0,C 180,E1 -14456.793,E2 -14456.793} C_VEL
LIN {X 0,Y 333.685,Z 385.052,A -85,B 0,C 180,E1 -14457.844,E2 -14457.844} C_VEL
LIN {X 0,Y 336.378,Z 396.837,A -85,B 0,C 180,E1 -14461.28,E2 -14461.28} C_VEL
LIN {X 0,Y 338.009,Z 405.297,A -85,B 0,C 180,E1 -14463.631,E2 -14463.631} C_VEL
LIN {X 0,Y 338.203,Z 408.435,A -85,B 0,C 180,E1 -14464.457,E2 -14464.457} C_VEL
LIN {X 0,Y 337.406,Z 414.7,A -85,B 0,C 180,E1 -14466.021,E2 -14466.021} C_VEL
LIN {X 0,Y 342.502,Z 444.634,A -85,B 0,C 180,E1 -14467.065,E2 -14467.065} C_VEL
LIN {X 0,Y 343.724,Z 453.972,A -85,B 0,C 180,E1 -14467.357,E2 -14467.357} C_VEL
LIN {X 0,Y 342.353,Z 523.287,A -85,B 0,C 180,E1 -14468.828,E2 -14468.828} C_VEL
LIN {X 0,Y 341.557,Z 536.48,A -85,B 0,C 180,E1 -14469.329,E2 -14469.329} C_VEL
LIN {X 0,Y 340.472,Z 549.72,A -85,B 0,C 180,E1 -14470.088,E2 -14470.088} C_VEL
LIN {X 0,Y 339.353,Z 560.846,A -85,B 0,C 180,E1 -14470.963,E2 -14470.963} C_VEL
LIN {X 0,Y 337.957,Z 572.434,A -85,B 0,C 180,E1 -14472.138,E2 -14472.138} C_VEL
LIN {X 0,Y 336.557,Z 583.194,A -85,B 0,C 180,E1 -14473.517,E2 -14473.517} C_VEL
LIN {X 0,Y 335.565,Z 591.741,A -85,B 0,C 180,E1 -14474.88,E2 -14474.88} C_VEL
LIN {X 0,Y 334.422,Z 600.682,A -85,B 0,C 180,E1 -14476.634,E2 -14476.634} C_VEL
LIN {X 0,Y 333.362,Z 608.125,A -85,B 0,C 180,E1 -14478.447,E2 -14478.447} C_VEL
LIN {X 0,Y 332.741,Z 614.114,A -85,B 0,C 180,E1 -14480.272,E2 -14480.272} C_VEL
LIN {X 0,Y 332.318,Z 618.848,A -85,B 0,C 180,E1 -14482.099,E2 -14482.099} C_VEL
LIN {X 0,Y 332.031,Z 622.903,A -85,B 0,C 180,E1 -14484.176,E2 -14484.176} C_VEL
LIN {X 0,Y 331.998,Z 625.738,A -85,B 0,C 180,E1 -14486.359,E2 -14486.359} C_VEL
LIN {X 0,Y 331.987,Z 627.349,A -85,B 0,C 180,E1 -14488.787,E2 -14488.787} C_VEL
LIN {X 0,Y 332.043,Z 627.566,A -85,B 0,C 180,E1 -14490,E2 -14490} C_VEL
LIN {X 0,Y 331.987,Z 627.344,A -85,B 0,C 180,E1 -14491.213,E2 -14491.213} C_VEL
LIN {X 0,Y 331.998,Z 625.727,A -85,B 0,C 180,E1 -14493.641,E2 -14493.641} C_VEL
LIN {X 0,Y 332.009,Z 622.941,A -85,B 0,C 180,E1 -14495.787,E2 -14495.787} C_VEL
LIN {X 0,Y 332.317,Z 618.81,A -85,B 0,C 180,E1 -14497.901,E2 -14497.901} C_VEL
LIN {X 0,Y 332.735,Z 614.066,A -85,B 0,C 180,E1 -14499.728,E2 -14499.728} C_VEL
LIN {X 0,Y 333.503,Z 606.944,A -85,B 0,C 180,E1 -14501.856,E2 -14501.856} C_VEL
LIN {X 0,Y 334.629,Z 599.226,A -85,B 0,C 180,E1 -14503.667,E2 -14503.667} C_VEL
LIN {X 0,Y 335.636,Z 591.414,A -85,B 0,C 180,E1 -14505.157,E2 -14505.157} C_VEL
LIN {X 0,Y 336.731,Z 581.898,A -85,B 0,C 180,E1 -14506.646,E2 -14506.646} C_VEL
LIN {X 0,Y 338.159,Z 571,A -85,B 0,C 180,E1 -14508.007,E2 -14508.007} C_VEL
LIN {X 0,Y 339.313,Z 560.673,A -85,B 0,C 180,E1 -14509.039,E2 -14509.039} C_VEL
LIN {X 0,Y 340.535,Z 548.344,A -85,B 0,C 180,E1 -14509.987,E2 -14509.987} C_VEL
LIN {X 0,Y 341.599,Z 535.367,A -85,B 0,C 180,E1 -14510.708,E2 -14510.708} C_VEL
LIN {X 0,Y 342.309,Z 522.763,A -85,B 0,C 180,E1 -14511.175,E2 -14511.175} C_VEL
LIN {X 0,Y 343.669,Z 452.985,A -85,B 0,C 180,E1 -14512.65,E2 -14512.65} C_VEL
LIN {X 0,Y 339.025,Z 423.788,A -85,B 0,C 180,E1 -14513.632,E2 -14513.632} C_VEL
LIN {X 0,Y 337.422,Z 414.64,A -85,B 0,C 180,E1 -14513.977,E2 -14513.977} C_VEL
LIN {X 0,Y 338.234,Z 407.08,A -85,B 0,C 180,E1 -14515.87,E2 -14515.87} C_VEL
LIN {X 0,Y 336.376,Z 396.738,A -85,B 0,C 180,E1 -14518.72,E2 -14518.72} C_VEL
LIN {X 0,Y 333.649,Z 384.927,A -85,B 0,C 180,E1 -14522.195,E2 -14522.195} C_VEL
LIN {X 0,Y 333.676,Z 384.921,A -85,B 0,C 180,E1 -14526.138,E2 -14526.138} C_VEL
LIN {X 0,Y 333.666,Z 384.922,A -85,B 0,C 180,E1 -14529.189,E2 -14529.189} C_VEL
LIN {X 0,Y 333.634,Z 384.923,A -85,B 0,C 180,E1 -14532.5,E2 -14532.5} C_VEL
LIN {X 0,Y 333.671,Z 384.919,A -85,B 0,C 180,E1 -14535.967,E2 -14535.967} C_VEL
LIN {X 0,Y 333.698,Z 384.919,A -85,B 0,C 180,E1 -14539.304,E2 -14539.304} C_VEL
LIN {X 0,Y 333.661,Z 384.922,A -85,B 0,C 180,E1 -14543.167,E2 -14543.167} C_VEL
LIN {X 0,Y 333.631,Z 384.923,A -85,B 0,C 180,E1 -14546.791,E2 -14546.791} C_VEL
LIN {X 0,Y 333.697,Z 384.917,A -85,B 0,C 180,E1 -14549.71,E2 -14549.71} C_VEL
LIN {X 0,Y 333.739,Z 384.909,A -85,B 0,C 180,E1 -14552.401,E2 -14552.401} C_VEL
LIN {X 0,Y 333.721,Z 384.916,A -85,B 0,C 180,E1 -14555.09,E2 -14555.09} C_VEL
LIN {X 0,Y 333.674,Z 384.921,A -85,B 0,C 180,E1 -14559.019,E2 -14559.019} C_VEL
LIN {X 0,Y 333.787,Z 384.904,A -85,B 0,C 180,E1 -14561.589,E2 -14561.589} C_VEL
LIN {X 0,Y 333.802,Z 384.904,A -85,B 0,C 180,E1 -14565.576,E2 -14565.576} C_VEL
LIN {X 0,Y 333.831,Z 384.901,A -85,B 0,C 180,E1 -14569.078,E2 -14569.078} C_VEL
LIN {X 0,Y 334.018,Z 384.878,A -85,B 0,C 180,E1 -14572.747,E2 -14572.747} C_VEL
LIN {X 0,Y 333.806,Z 384.904,A -85,B 0,C 180,E1 -14575.169,E2 -14575.169} C_VEL
LIN {X 0,Y 334.1,Z 384.863,A -85,B 0,C 180,E1 -14577.589,E2 -14577.589} C_VEL
LIN {X 0,Y 334.26,Z 384.845,A -85,B 0,C 180,E1 -14580,E2 -14580} C_VEL
LIN {X 0,Y 334.101,Z 384.866,A -85,B 0,C 180,E1 -14582.411,E2 -14582.411} C_VEL
LIN {X 0,Y 334.018,Z 384.877,A -85,B 0,C 180,E1 -14587.253,E2 -14587.253} C_VEL
LIN {X 0,Y 333.83,Z 384.9,A -85,B 0,C 180,E1 -14590.922,E2 -14590.922} C_VEL
LIN {X 0,Y 333.802,Z 384.906,A -85,B 0,C 180,E1 -14594.635,E2 -14594.635} C_VEL
LIN {X 0,Y 333.791,Z 384.906,A -85,B 0,C 180,E1 -14598.656,E2 -14598.656} C_VEL
LIN {X 0,Y 333.686,Z 384.919,A -85,B 0,C 180,E1 -14602.279,E2 -14602.279} C_VEL
LIN {X 0,Y 333.73,Z 384.911,A -85,B 0,C 180,E1 -14606.247,E2 -14606.247} C_VEL
LIN {X 0,Y 333.705,Z 384.916,A -85,B 0,C 180,E1 -14608.973,E2 -14608.973} C_VEL
LIN {X 0,Y 333.638,Z 384.927,A -85,B 0,C 180,E1 -14612.588,E2 -14612.588} C_VEL
LIN {X 0,Y 333.672,Z 384.921,A -85,B 0,C 180,E1 -14616.14,E2 -14616.14} C_VEL
LIN {X 0,Y 333.681,Z 384.918,A -85,B 0,C 180,E1 -14619.188,E2 -14619.188} C_VEL
LIN {X 0,Y 333.687,Z 384.921,A -85,B 0,C 180,E1 -14622.512,E2 -14622.512} C_VEL
LIN {X 0,Y 333.632,Z 384.925,A -85,B 0,C 180,E1 -14625.962,E2 -14625.962} C_VEL
LIN {X 0,Y 333.645,Z 384.922,A -85,B 0,C 180,E1 -14629.316,E2 -14629.316} C_VEL
LIN {X 0,Y 333.666,Z 384.92,A -85,B 0,C 180,E1 -14633.168,E2 -14633.168} C_VEL
LIN {X 0,Y 333.638,Z 384.924,A -85,B 0,C 180,E1 -14636.793,E2 -14636.793} C_VEL
LIN {X 0,Y 333.694,Z 384.919,A -85,B 0,C 180,E1 -14639.713,E2 -14639.713} C_VEL
LIN {X 0,Y 333.773,Z 385.007,A -85,B 0,C 180,E1 -14643.505,E2 -14643.505} C_VEL
LIN {X 0,Y 335.328,Z 392.572,A -85,B 0,C 180,E1 -14645.953,E2 -14645.953} C_VEL
LIN {X 0,Y 342.352,Z 410.642,A -85,B 0,C 180,E1 -14646.889,E2 -14646.889} C_VEL
LIN {X 0,Y 344.349,Z 421.013,A -85,B 0,C 180,E1 -14647.263,E2 -14647.263} C_VEL
LIN {X 0,Y 342.72,Z 499.701,A -85,B 0,C 180,E1 -14648.931,E2 -14648.931} C_VEL
LIN {X 0,Y 342.028,Z 512.706,A -85,B 0,C 180,E1 -14649.437,E2 -14649.437} C_VEL
LIN {X 0,Y 341.266,Z 524.706,A -85,B 0,C 180,E1 -14650.136,E2 -14650.136} C_VEL
LIN {X 0,Y 340.271,Z 536.034,A -85,B 0,C 180,E1 -14651.017,E2 -14651.017} C_VEL
LIN {X 0,Y 339.044,Z 547.534,A -85,B 0,C 180,E1 -14652.18,E2 -14652.18} C_VEL
LIN {X 0,Y 337.956,Z 558.108,A -85,B 0,C 180,E1 -14653.541,E2 -14653.541} C_VEL
LIN {X 0,Y 336.755,Z 566.643,A -85,B 0,C 180,E1 -14654.879,E2 -14654.879} C_VEL
LIN {X 0,Y 335.67,Z 574.5,A -85,B 0,C 180,E1 -14656.377,E2 -14656.377} C_VEL
LIN {X 0,Y 334.556,Z 582.177,A -85,B 0,C 180,E1 -14658.181,E2 -14658.181} C_VEL
LIN {X 0,Y 333.565,Z 589.22,A -85,B 0,C 180,E1 -14660.296,E2 -14660.296} C_VEL
LIN {X 0,Y 332.913,Z 593.911,A -85,B 0,C 180,E1 -14662.113,E2 -14662.113} C_VEL
LIN {X 0,Y 332.591,Z 597.494,A -85,B 0,C 180,E1 -14663.935,E2 -14663.935} C_VEL
LIN {X 0,Y 332.378,Z 599.347,A -85,B 0,C 180,E1 -14665.148,E2 -14665.148} C_VEL
LIN {X 0,Y 332.185,Z 600.743,A -85,B 0,C 180,E1 -14666.361,E2 -14666.361} C_VEL
LIN {X 0,Y 332.044,Z 602.344,A -85,B 0,C 180,E1 -14668.787,E2 -14668.787} C_VEL
LIN {X 0,Y 332.048,Z 602.575,A -85,B 0,C 180,E1 -14670,E2 -14670} C_VEL
LIN {X 0,Y 332.044,Z 602.385,A -85,B 0,C 180,E1 -14671.213,E2 -14671.213} C_VEL
LIN {X 0,Y 332.184,Z 600.837,A -85,B 0,C 180,E1 -14673.639,E2 -14673.639} C_VEL
LIN {X 0,Y 332.376,Z 599.482,A -85,B 0,C 180,E1 -14674.852,E2 -14674.852} C_VEL
LIN {X 0,Y 332.79,Z 596.016,A -85,B 0,C 180,E1 -14676.989,E2 -14676.989} C_VEL
LIN {X 0,Y 333.31,Z 591.191,A -85,B 0,C 180,E1 -14679.099,E2 -14679.099} C_VEL
LIN {X 0,Y 334.219,Z 584.764,A -85,B 0,C 180,E1 -14681.216,E2 -14681.216} C_VEL
LIN {X 0,Y 335.209,Z 577.7,A -85,B 0,C 180,E1 -14683.025,E2 -14683.025} C_VEL
LIN {X 0,Y 336.463,Z 568.894,A -85,B 0,C 180,E1 -14684.825,E2 -14684.825} C_VEL
LIN {X 0,Y 337.708,Z 559.88,A -85,B 0,C 180,E1 -14686.312,E2 -14686.312} C_VEL
LIN {X 0,Y 338.768,Z 550.224,A -85,B 0,C 180,E1 -14687.615,E2 -14687.615} C_VEL
LIN {X 0,Y 339.865,Z 540.277,A -85,B 0,C 180,E1 -14688.694,E2 -14688.694} C_VEL
LIN {X 0,Y 341.028,Z 528.169,A -85,B 0,C 180,E1 -14689.722,E2 -14689.722} C_VEL
LIN {X 0,Y 341.938,Z 515.479,A -85,B 0,C 180,E1 -14690.529,E2 -14690.529} C_VEL
LIN {X 0,Y 342.651,Z 502.828,A -85,B 0,C 180,E1 -14691.074,E2 -14691.074} C_VEL
LIN {X 0,Y 342.998,Z 484.886,A -85,B 0,C 180,E1 -14691.524,E2 -14691.524} C_VEL
LIN {X 0,Y 344.281,Z 419.931,A -85,B 0,C 180,E1 -14692.874,E2 -14692.874} C_VEL
LIN {X 0,Y 342.045,Z 409.933,A -85,B 0,C 180,E1 -14693.258,E2 -14693.258} C_VEL
LIN {X 0,Y 335.279,Z 392.287,A -85,B 0,C 180,E1 -14694.194,E2 -14694.194} C_VEL
LIN {X 0,Y 333.817,Z 385.155,A -85,B 0,C 180,E1 -14696.553,E2 -14696.553} C_VEL
LIN {X 0,Y 333.216,Z 384.977,A -85,B 0,C 180,E1 -14697.171,E2 -14697.171} C_VEL
LIN {X 0,Y 329.838,Z 385.398,A -85,B 0,C 180,E1 -14699.12,E2 -14699.12} C_VEL
LIN {X 0,Y 327.572,Z 385.878,A -85,B 0,C 180,E1 -14700.483,E2 -14700.483} C_VEL
LIN {X 0,Y 326.641,Z 385.813,A -85,B 0,C 180,E1 -14701.54,E2 -14701.54} C_VEL
LIN {X 0,Y 326.575,Z 385.8,A -85,B 0,C 180,E1 -14701.896,E2 -14701.896} C_VEL
LIN {X 0,Y 326.612,Z 385.801,A -85,B 0,C 180,E1 -14705.519,E2 -14705.519} C_VEL
LIN {X 0,Y 326.61,Z 385.799,A -85,B 0,C 180,E1 -14709.226,E2 -14709.226} C_VEL
LIN {X 0,Y 326.583,Z 385.801,A -85,B 0,C 180,E1 -14712.973,E2 -14712.973} C_VEL
LIN {X 0,Y 326.626,Z 385.793,A -85,B 0,C 180,E1 -14717.017,E2 -14717.017} C_VEL
LIN {X 0,Y 326.641,Z 385.794,A -85,B 0,C 180,E1 -14720.765,E2 -14720.765} C_VEL
LIN {X 0,Y 326.608,Z 385.799,A -85,B 0,C 180,E1 -14724.48,E2 -14724.48} C_VEL
LIN {X 0,Y 326.605,Z 385.801,A -85,B 0,C 180,E1 -14727.455,E2 -14727.455} C_VEL
LIN {X 0,Y 326.655,Z 385.792,A -85,B 0,C 180,E1 -14730.34,E2 -14730.34} C_VEL
LIN {X 0,Y 326.685,Z 385.789,A -85,B 0,C 180,E1 -14734.516,E2 -14734.516} C_VEL
LIN {X 0,Y 326.641,Z 385.794,A -85,B 0,C 180,E1 -14738.545,E2 -14738.545} C_VEL
LIN {X 0,Y 326.738,Z 385.786,A -85,B 0,C 180,E1 -14741.177,E2 -14741.177} C_VEL
LIN {X 0,Y 326.757,Z 385.784,A -85,B 0,C 180,E1 -14745.433,E2 -14745.433} C_VEL
LIN {X 0,Y 326.766,Z 385.778,A -85,B 0,C 180,E1 -14748.839,E2 -14748.839} C_VEL
LIN {X 0,Y 326.972,Z 385.754,A -85,B 0,C 180,E1 -14752.59,E2 -14752.59} C_VEL
LIN {X 0,Y 326.773,Z 385.78,A -85,B 0,C 180,E1 -14755.065,E2 -14755.065} C_VEL
LIN {X 0,Y 327.041,Z 385.746,A -85,B 0,C 180,E1 -14757.537,E2 -14757.537} C_VEL
LIN {X 0,Y 327.211,Z 385.723,A -85,B 0,C 180,E1 -14760,E2 -14760} C_VEL
LIN {X 0,Y 327.042,Z 385.741,A -85,B 0,C 180,E1 -14762.463,E2 -14762.463} C_VEL
LIN {X 0,Y 326.989,Z 385.751,A -85,B 0,C 180,E1 -14766.169,E2 -14766.169} C_VEL
LIN {X 0,Y 326.908,Z 385.761,A -85,B 0,C 180,E1 -14768.655,E2 -14768.655} C_VEL
LIN {X 0,Y 326.732,Z 385.784,A -85,B 0,C 180,E1 -14772.421,E2 -14772.421} C_VEL
LIN {X 0,Y 326.748,Z 385.784,A -85,B 0,C 180,E1 -14774.958,E2 -14774.958} C_VEL
LIN {X 0,Y 326.726,Z 385.787,A -85,B 0,C 180,E1 -14778.838,E2 -14778.838} C_VEL
LIN {X 0,Y 326.615,Z 385.803,A -85,B 0,C 180,E1 -14782.788,E2 -14782.788} C_VEL
LIN {X 0,Y 326.684,Z 385.789,A -85,B 0,C 180,E1 -14785.484,E2 -14785.484} C_VEL
LIN {X 0,Y 326.655,Z 385.792,A -85,B 0,C 180,E1 -14789.66,E2 -14789.66} C_VEL
LIN {X 0,Y 326.602,Z 385.798,A -85,B 0,C 180,E1 -14794.02,E2 -14794.02} C_VEL
LIN {X 0,Y 326.625,Z 385.795,A -85,B 0,C 180,E1 -14797.24,E2 -14797.24} C_VEL
LIN {X 0,Y 326.631,Z 385.797,A -85,B 0,C 180,E1 -14800.203,E2 -14800.203} C_VEL
LIN {X 0,Y 326.619,Z 385.795,A -85,B 0,C 180,E1 -14803.516,E2 -14803.516} C_VEL
LIN {X 0,Y 326.585,Z 385.803,A -85,B 0,C 180,E1 -14807.027,E2 -14807.027} C_VEL
LIN {X 0,Y 326.627,Z 385.799,A -85,B 0,C 180,E1 -14810.77,E2 -14810.77} C_VEL
LIN {X 0,Y 326.612,Z 385.804,A -85,B 0,C 180,E1 -14814.481,E2 -14814.481} C_VEL
LIN {X 0,Y 326.635,Z 385.92,A -85,B 0,C 180,E1 -14817.388,E2 -14817.388} C_VEL
LIN {X 0,Y 329.082,Z 396.557,A -85,B 0,C 180,E1 -14820.582,E2 -14820.582} C_VEL
LIN {X 0,Y 331.123,Z 406.879,A -85,B 0,C 180,E1 -14823.531,E2 -14823.531} C_VEL
LIN {X 0,Y 331.181,Z 410.7,A -85,B 0,C 180,E1 -14824.55,E2 -14824.55} C_VEL
LIN {X 0,Y 330.678,Z 414.39,A -85,B 0,C 180,E1 -14825.491,E2 -14825.491} C_VEL
LIN {X 0,Y 336.01,Z 445.827,A -85,B 0,C 180,E1 -14826.629,E2 -14826.629} C_VEL
LIN {X 0,Y 337.17,Z 455.003,A -85,B 0,C 180,E1 -14826.921,E2 -14826.921} C_VEL
LIN {X 0,Y 335.753,Z 523.033,A -85,B 0,C 180,E1 -14828.391,E2 -14828.391} C_VEL
LIN {X 0,Y 334.931,Z 536.222,A -85,B 0,C 180,E1 -14828.901,E2 -14828.901} C_VEL
LIN {X 0,Y 333.807,Z 549.459,A -85,B 0,C 180,E1 -14829.673,E2 -14829.673} C_VEL
LIN {X 0,Y 332.617,Z 560.582,A -85,B 0,C 180,E1 -14830.562,E2 -14830.562} C_VEL
LIN {X 0,Y 331.197,Z 572.17,A -85,B 0,C 180,E1 -14831.761,E2 -14831.761} C_VEL
LIN {X 0,Y 329.77,Z 582.607,A -85,B 0,C 180,E1 -14833.12,E2 -14833.12} C_VEL
LIN {X 0,Y 328.646,Z 591.808,A -85,B 0,C 180,E1 -14834.616,E2 -14834.616} C_VEL
LIN {X 0,Y 327.487,Z 600.415,A -85,B 0,C 180,E1 -14836.346,E2 -14836.346} C_VEL
LIN {X 0,Y 326.383,Z 607.859,A -85,B 0,C 180,E1 -14838.196,E2 -14838.196} C_VEL
LIN {X 0,Y 325.706,Z 613.846,A -85,B 0,C 180,E1 -14840.06,E2 -14840.06} C_VEL
LIN {X 0,Y 325.245,Z 618.58,A -85,B 0,C 180,E1 -14841.926,E2 -14841.926} C_VEL
LIN {X 0,Y 324.997,Z 622.2,A -85,B 0,C 180,E1 -14843.793,E2 -14843.793} C_VEL
LIN {X 0,Y 324.896,Z 624.068,A -85,B 0,C 180,E1 -14845.036,E2 -14845.036} C_VEL
LIN {X 0,Y 324.902,Z 625.471,A -85,B 0,C 180,E1 -14846.279,E2 -14846.279} C_VEL
LIN {X 0,Y 324.892,Z 627.082,A -85,B 0,C 180,E1 -14848.761,E2 -14848.761} C_VEL
LIN {X 0,Y 324.948,Z 627.299,A -85,B 0,C 180,E1 -14850,E2 -14850} C_VEL
LIN {X 0,Y 324.892,Z 627.076,A -85,B 0,C 180,E1 -14851.239,E2 -14851.239} C_VEL
LIN {X 0,Y 324.901,Z 625.459,A -85,B 0,C 180,E1 -14853.721,E2 -14853.721} C_VEL
LIN {X 0,Y 324.914,Z 622.939,A -85,B 0,C 180,E1 -14855.732,E2 -14855.732} C_VEL
LIN {X 0,Y 325.146,Z 619.862,A -85,B 0,C 180,E1 -14857.451,E2 -14857.451} C_VEL
LIN {X 0,Y 325.533,Z 615.501,A -85,B 0,C 180,E1 -14859.318,E2 -14859.318} C_VEL
LIN {X 0,Y 326.106,Z 609.949,A -85,B 0,C 180,E1 -14861.184,E2 -14861.184} C_VEL
LIN {X 0,Y 327.063,Z 603.029,A -85,B 0,C 180,E1 -14863.039,E2 -14863.039} C_VEL
LIN {X 0,Y 328.035,Z 595.966,A -85,B 0,C 180,E1 -14864.58,E2 -14864.58} C_VEL
LIN {X 0,Y 329.193,Z 587.455,A -85,B 0,C 180,E1 -14866.113,E2 -14866.113} C_VEL
LIN {X 0,Y 330.542,Z 576.944,A -85,B 0,C 180,E1 -14867.636,E2 -14867.636} C_VEL
LIN {X 0,Y 332.081,Z 565.122,A -85,B 0,C 180,E1 -14868.989,E2 -14868.989} C_VEL
LIN {X 0,Y 333.386,Z 553.222,A -85,B 0,C 180,E1 -14870.032,E2 -14870.032} C_VEL
LIN {X 0,Y 334.534,Z 540.843,A -85,B 0,C 180,E1 -14870.844,E2 -14870.844} C_VEL
LIN {X 0,Y 335.437,Z 528.113,A -85,B 0,C 180,E1 -14871.428,E2 -14871.428} C_VEL
LIN {X 0,Y 335.96,Z 514.704,A -85,B 0,C 180,E1 -14871.796,E2 -14871.796} C_VEL
LIN {X 0,Y 337.03,Z 453.172,A -85,B 0,C 180,E1 -14873.111,E2 -14873.111} C_VEL
LIN {X 0,Y 332.033,Z 421.969,A -85,B 0,C 180,E1 -14874.196,E2 -14874.196} C_VEL
LIN {X 0,Y 330.64,Z 414.419,A -85,B 0,C 180,E1 -14874.487,E2 -14874.487} C_VEL
LIN {X 0,Y 331.269,Z 408.078,A -85,B 0,C 180,E1 -14876.117,E2 -14876.117} C_VEL
LIN {X 0,Y 329.392,Z 397.969,A -85,B 0,C 180,E1 -14878.98,E2 -14878.98} C_VEL
LIN {X 0,Y 326.973,Z 387.391,A -85,B 0,C 180,E1 -14882.138,E2 -14882.138} C_VEL
LIN {X 0,Y 326.617,Z 385.805,A -85,B 0,C 180,E1 -14882.685,E2 -14882.685} C_VEL
LIN {X 0,Y 326.612,Z 385.804,A -85,B 0,C 180,E1 -14885.519,E2 -14885.519} C_VEL
LIN {X 0,Y 326.627,Z 385.799,A -85,B 0,C 180,E1 -14889.23,E2 -14889.23} C_VEL
LIN {X 0,Y 326.583,Z 385.805,A -85,B 0,C 180,E1 -14893.521,E2 -14893.521} C_VEL
LIN {X 0,Y 326.626,Z 385.796,A -85,B 0,C 180,E1 -14897.017,E2 -14897.017} C_VEL
LIN {X 0,Y 326.641,Z 385.795,A -85,B 0,C 180,E1 -14900.765,E2 -14900.765} C_VEL
LIN {X 0,Y 326.608,Z 385.799,A -85,B 0,C 180,E1 -14904.48,E2 -14904.48} C_VEL
LIN {X 0,Y 326.602,Z 385.803,A -85,B 0,C 180,E1 -14907.455,E2 -14907.455} C_VEL
LIN {X 0,Y 326.655,Z 385.791,A -85,B 0,C 180,E1 -14910.34,E2 -14910.34} C_VEL
LIN {X 0,Y 326.684,Z 385.789,A -85,B 0,C 180,E1 -14914.516,E2 -14914.516} C_VEL
LIN {X 0,Y 326.64,Z 385.794,A -85,B 0,C 180,E1 -14918.545,E2 -14918.545} C_VEL
LIN {X 0,Y 326.738,Z 385.786,A -85,B 0,C 180,E1 -14921.177,E2 -14921.177} C_VEL
LIN {X 0,Y 326.756,Z 385.783,A -85,B 0,C 180,E1 -14925.433,E2 -14925.433} C_VEL
LIN {X 0,Y 326.766,Z 385.781,A -85,B 0,C 180,E1 -14928.839,E2 -14928.839} C_VEL
LIN {X 0,Y 326.972,Z 385.754,A -85,B 0,C 180,E1 -14932.59,E2 -14932.59} C_VEL
LIN {X 0,Y 326.773,Z 385.781,A -85,B 0,C 180,E1 -14935.065,E2 -14935.065} C_VEL
LIN {X 0,Y 327.041,Z 385.742,A -85,B 0,C 180,E1 -14937.537,E2 -14937.537} C_VEL
LIN {X 0,Y 327.211,Z 385.723,A -85,B 0,C 180,E1 -14940,E2 -14940} C_VEL
LIN {X 0,Y 327.041,Z 385.746,A -85,B 0,C 180,E1 -14942.463,E2 -14942.463} C_VEL
LIN {X 0,Y 326.964,Z 385.751,A -85,B 0,C 180,E1 -14946.684,E2 -14946.684} C_VEL
LIN {X 0,Y 326.809,Z 385.773,A -85,B 0,C 180,E1 -14949.907,E2 -14949.907} C_VEL
LIN {X 0,Y 326.754,Z 385.779,A -85,B 0,C 180,E1 -14953.686,E2 -14953.686} C_VEL
LIN {X 0,Y 326.693,Z 385.787,A -85,B 0,C 180,E1 -14957.528,E2 -14957.528} C_VEL
LIN {X 0,Y 326.659,Z 385.789,A -85,B 0,C 180,E1 -14960.135,E2 -14960.135} C_VEL
LIN {X 0,Y 326.646,Z 385.795,A -85,B 0,C 180,E1 -14964.129,E2 -14964.129} C_VEL
LIN {X 0,Y 326.679,Z 385.792,A -85,B 0,C 180,E1 -14966.858,E2 -14966.858} C_VEL
LIN {X 0,Y 326.634,Z 385.797,A -85,B 0,C 180,E1 -14970.612,E2 -14970.612} C_VEL
LIN {X 0,Y 326.602,Z 385.801,A -85,B 0,C 180,E1 -14974.02,E2 -14974.02} C_VEL
LIN {X 0,Y 326.625,Z 385.795,A -85,B 0,C 180,E1 -14977.24,E2 -14977.24} C_VEL
LIN {X 0,Y 326.632,Z 385.799,A -85,B 0,C 180,E1 -14980.203,E2 -14980.203} C_VEL
LIN {X 0,Y 326.619,Z 385.797,A -85,B 0,C 180,E1 -14983.516,E2 -14983.516} C_VEL
LIN {X 0,Y 326.583,Z 385.802,A -85,B 0,C 180,E1 -14987.027,E2 -14987.027} C_VEL
LIN {X 0,Y 326.61,Z 385.8,A -85,B 0,C 180,E1 -14990.773,E2 -14990.773} C_VEL
LIN {X 0,Y 326.612,Z 385.802,A -85,B 0,C 180,E1 -14994.481,E2 -14994.481} C_VEL
LIN {X 0,Y 326.609,Z 385.8,A -85,B 0,C 180,E1 -14997.457,E2 -14997.457} C_VEL
LIN {X 0,Y 326.648,Z 385.796,A -85,B 0,C 180,E1 -15000.34,E2 -15000.34} C_VEL
LIN {X 0,Y 326.735,Z 385.81,A -85,B 0,C 180,E1 -15003.061,E2 -15003.061} C_VEL
LIN {X 0,Y 328.118,Z 392.578,A -85,B 0,C 180,E1 -15005.362,E2 -15005.362} C_VEL
LIN {X 0,Y 336.149,Z 413.381,A -85,B 0,C 180,E1 -15006.493,E2 -15006.493} C_VEL
LIN {X 0,Y 337.821,Z 421.308,A -85,B 0,C 180,E1 -15006.798,E2 -15006.798} C_VEL
LIN {X 0,Y 336.106,Z 499.984,A -85,B 0,C 180,E1 -15008.496,E2 -15008.496} C_VEL
LIN {X 0,Y 335.387,Z 512.983,A -85,B 0,C 180,E1 -15009.011,E2 -15009.011} C_VEL
LIN {X 0,Y 334.618,Z 524.98,A -85,B 0,C 180,E1 -15009.724,E2 -15009.724} C_VEL
LIN {X 0,Y 333.583,Z 536.306,A -85,B 0,C 180,E1 -15010.621,E2 -15010.621} C_VEL
LIN {X 0,Y 332.259,Z 548.2,A -85,B 0,C 180,E1 -15011.853,E2 -15011.853} C_VEL
LIN {X 0,Y 331.164,Z 558.379,A -85,B 0,C 180,E1 -15013.193,E2 -15013.193} C_VEL
LIN {X 0,Y 329.92,Z 566.913,A -85,B 0,C 180,E1 -15014.558,E2 -15014.558} C_VEL
LIN {X 0,Y 328.755,Z 574.77,A -85,B 0,C 180,E1 -15016.084,E2 -15016.084} C_VEL
LIN {X 0,Y 327.617,Z 582.446,A -85,B 0,C 180,E1 -15017.927,E2 -15017.927} C_VEL
LIN {X 0,Y 326.561,Z 589.489,A -85,B 0,C 180,E1 -15020.086,E2 -15020.086} C_VEL
LIN {X 0,Y 325.875,Z 594.179,A -85,B 0,C 180,E1 -15021.942,E2 -15021.942} C_VEL
LIN {X 0,Y 325.537,Z 597.762,A -85,B 0,C 180,E1 -15023.803,E2 -15023.803} C_VEL
LIN {X 0,Y 325.326,Z 599.615,A -85,B 0,C 180,E1 -15025.043,E2 -15025.043} C_VEL
LIN {X 0,Y 325.116,Z 601.01,A -85,B 0,C 180,E1 -15026.282,E2 -15026.282} C_VEL
LIN {X 0,Y 324.95,Z 602.612,A -85,B 0,C 180,E1 -15028.761,E2 -15028.761} C_VEL
LIN {X 0,Y 324.954,Z 602.842,A -85,B 0,C 180,E1 -15030,E2 -15030} C_VEL
LIN {X 0,Y 324.95,Z 602.652,A -85,B 0,C 180,E1 -15031.239,E2 -15031.239} C_VEL
LIN {X 0,Y 325.115,Z 601.103,A -85,B 0,C 180,E1 -15033.718,E2 -15033.718} C_VEL
LIN {X 0,Y 325.325,Z 599.748,A -85,B 0,C 180,E1 -15034.957,E2 -15034.957} C_VEL
LIN {X 0,Y 325.703,Z 596.599,A -85,B 0,C 180,E1 -15036.979,E2 -15036.979} C_VEL
LIN {X 0,Y 326.298,Z 591.457,A -85,B 0,C 180,E1 -15039.296,E2 -15039.296} C_VEL
LIN {X 0,Y 327.231,Z 585.031,A -85,B 0,C 180,E1 -15041.459,E2 -15041.459} C_VEL
LIN {X 0,Y 328.267,Z 577.966,A -85,B 0,C 180,E1 -15043.306,E2 -15043.306} C_VEL
LIN {X 0,Y 329.602,Z 569.158,A -85,B 0,C 180,E1 -15045.141,E2 -15045.141} C_VEL
LIN {X 0,Y 331.02,Z 559.344,A -85,B 0,C 180,E1 -15046.779,E2 -15046.779} C_VEL
LIN {X 0,Y 332.158,Z 549.078,A -85,B 0,C 180,E1 -15048.153,E2 -15048.153} C_VEL
LIN {X 0,Y 333.49,Z 537.386,A -85,B 0,C 180,E1 -15049.385,E2 -15049.385} C_VEL
LIN {X 0,Y 334.637,Z 525.394,A -85,B 0,C 180,E1 -15050.355,E2 -15050.355} C_VEL
LIN {X 0,Y 335.516,Z 512.017,A -85,B 0,C 180,E1 -15051.141,E2 -15051.141} C_VEL
LIN {X 0,Y 336.228,Z 498.448,A -85,B 0,C 180,E1 -15051.657,E2 -15051.657} C_VEL
LIN {X 0,Y 337.786,Z 421.163,A -85,B 0,C 180,E1 -15053.317,E2 -15053.317} C_VEL
LIN {X 0,Y 335.853,Z 412.399,A -85,B 0,C 180,E1 -15053.662,E2 -15053.662} C_VEL
LIN {X 0,Y 328.133,Z 392.648,A -85,B 0,C 180,E1 -15054.732,E2 -15054.732} C_VEL
LIN {X 0,Y 326.719,Z 385.786,A -85,B 0,C 180,E1 -15057.113,E2 -15057.113} C_VEL
LIN {X 0,Y 326.589,Z 385.8,A -85,B 0,C 180,E1 -15061.095,E2 -15061.095} C_VEL
LIN {X 0,Y 326.575,Z 385.8,A -85,B 0,C 180,E1 -15061.896,E2 -15061.896} C_VEL
LIN {X 0,Y 325.923,Z 385.886,A -85,B 0,C 180,E1 -15062.927,E2 -15062.927} C_VEL
LIN {X 0,Y 323.058,Z 386.242,A -85,B 0,C 180,E1 -15064.603,E2 -15064.603} C_VEL
LIN {X 0,Y 320.637,Z 386.547,A -85,B 0,C 180,E1 -15065.962,E2 -15065.962} C_VEL
LIN {X 0,Y 319.625,Z 386.67,A -85,B 0,C 180,E1 -15067.014,E2 -15067.014} C_VEL
LIN {X 0,Y 319.559,Z 386.679,A -85,B 0,C 180,E1 -15067.37,E2 -15067.37} C_VEL
LIN {X 0,Y 319.527,Z 386.682,A -85,B 0,C 180,E1 -15071.287,E2 -15071.287} C_VEL
LIN {X 0,Y 319.54,Z 386.679,A -85,B 0,C 180,E1 -15074.732,E2 -15074.732} C_VEL
LIN {X 0,Y 319.594,Z 386.67,A -85,B 0,C 180,E1 -15078.388,E2 -15078.388} C_VEL
LIN {X 0,Y 319.594,Z 386.67,A -85,B 0,C 180,E1 -15082.339,E2 -15082.339} C_VEL
LIN {X 0,Y 319.556,Z 386.679,A -85,B 0,C 180,E1 -15085.123,E2 -15085.123} C_VEL
LIN {X 0,Y 319.566,Z 386.677,A -85,B 0,C 180,E1 -15089.057,E2 -15089.057} C_VEL
LIN {X 0,Y 319.603,Z 386.67,A -85,B 0,C 180,E1 -15092.497,E2 -15092.497} C_VEL
LIN {X 0,Y 319.6,Z 386.676,A -85,B 0,C 180,E1 -15095.303,E2 -15095.303} C_VEL
LIN {X 0,Y 319.591,Z 386.673,A -85,B 0,C 180,E1 -15098.047,E2 -15098.047} C_VEL
LIN {X 0,Y 319.683,Z 386.663,A -85,B 0,C 180,E1 -15100.962,E2 -15100.962} C_VEL
LIN {X 0,Y 319.725,Z 386.661,A -85,B 0,C 180,E1 -15105.276,E2 -15105.276} C_VEL
LIN {X 0,Y 319.753,Z 386.652,A -85,B 0,C 180,E1 -15109.873,E2 -15109.873} C_VEL
LIN {X 0,Y 319.926,Z 386.631,A -85,B 0,C 180,E1 -15112.426,E2 -15112.426} C_VEL
LIN {X 0,Y 319.742,Z 386.656,A -85,B 0,C 180,E1 -15114.956,E2 -15114.956} C_VEL
LIN {X 0,Y 319.985,Z 386.626,A -85,B 0,C 180,E1 -15117.482,E2 -15117.482} C_VEL
LIN {X 0,Y 320.162,Z 386.601,A -85,B 0,C 180,E1 -15120,E2 -15120} C_VEL
LIN {X 0,Y 319.985,Z 386.62,A -85,B 0,C 180,E1 -15122.518,E2 -15122.518} C_VEL
LIN {X 0,Y 319.945,Z 386.628,A -85,B 0,C 180,E1 -15126.306,E2 -15126.306} C_VEL
LIN {X 0,Y 319.836,Z 386.642,A -85,B 0,C 180,E1 -15128.848,E2 -15128.848} C_VEL
LIN {X 0,Y 319.679,Z 386.665,A -85,B 0,C 180,E1 -15132.7,E2 -15132.7} C_VEL
LIN {X 0,Y 319.693,Z 386.661,A -85,B 0,C 180,E1 -15135.296,E2 -15135.296} C_VEL
LIN {X 0,Y 319.668,Z 386.662,A -85,B 0,C 180,E1 -15139.255,E2 -15139.255} C_VEL
LIN {X 0,Y 319.564,Z 386.676,A -85,B 0,C 180,E1 -15143.32,E2 -15143.32} C_VEL
LIN {X 0,Y 319.629,Z 386.668,A -85,B 0,C 180,E1 -15146.089,E2 -15146.089} C_VEL
LIN {X 0,Y 319.584,Z 386.676,A -85,B 0,C 180,E1 -15148.934,E2 -15148.934} C_VEL
LIN {X 0,Y 319.527,Z 386.68,A -85,B 0,C 180,E1 -15151.862,E2 -15151.862} C_VEL
LIN {X 0,Y 319.575,Z 386.674,A -85,B 0,C 180,E1 -15155.544,E2 -15155.544} C_VEL
LIN {X 0,Y 319.58,Z 386.673,A -85,B 0,C 180,E1 -15158.007,E2 -15158.007} C_VEL
LIN {X 0,Y 319.593,Z 386.672,A -85,B 0,C 180,E1 -15161.612,E2 -15161.612} C_VEL
LIN {X 0,Y 319.564,Z 386.676,A -85,B 0,C 180,E1 -15165.272,E2 -15165.272} C_VEL
LIN {X 0,Y 319.53,Z 386.684,A -85,B 0,C 180,E1 -15168.713,E2 -15168.713} C_VEL
LIN {X 0,Y 319.577,Z 386.679,A -85,B 0,C 180,E1 -15172.345,E2 -15172.345} C_VEL
LIN {X 0,Y 319.559,Z 386.681,A -85,B 0,C 180,E1 -15175.124,E2 -15175.124} C_VEL
LIN {X 0,Y 319.588,Z 386.848,A -85,B 0,C 180,E1 -15176.925,E2 -15176.925} C_VEL
LIN {X 0,Y 322.215,Z 398.236,A -85,B 0,C 180,E1 -15180.437,E2 -15180.437} C_VEL
LIN {X 0,Y 324.132,Z 407.879,A -85,B 0,C 180,E1 -15183.263,E2 -15183.263} C_VEL
LIN {X 0,Y 324.296,Z 411.696,A -85,B 0,C 180,E1 -15184.315,E2 -15184.315} C_VEL
LIN {X 0,Y 323.929,Z 414.103,A -85,B 0,C 180,E1 -15184.941,E2 -15184.941} C_VEL
LIN {X 0,Y 329.088,Z 444.015,A -85,B 0,C 180,E1 -15186.071,E2 -15186.071} C_VEL
LIN {X 0,Y 330.611,Z 456.338,A -85,B 0,C 180,E1 -15186.472,E2 -15186.472} C_VEL
LIN {X 0,Y 329.176,Z 522.78,A -85,B 0,C 180,E1 -15187.937,E2 -15187.937} C_VEL
LIN {X 0,Y 328.329,Z 535.964,A -85,B 0,C 180,E1 -15188.455,E2 -15188.455} C_VEL
LIN {X 0,Y 327.252,Z 548.083,A -85,B 0,C 180,E1 -15189.165,E2 -15189.165} C_VEL
LIN {X 0,Y 325.913,Z 560.319,A -85,B 0,C 180,E1 -15190.146,E2 -15190.146} C_VEL
LIN {X 0,Y 324.431,Z 571.905,A -85,B 0,C 180,E1 -15191.366,E2 -15191.366} C_VEL
LIN {X 0,Y 322.953,Z 582.342,A -85,B 0,C 180,E1 -15192.753,E2 -15192.753} C_VEL
LIN {X 0,Y 321.731,Z 591.888,A -85,B 0,C 180,E1 -15194.345,E2 -15194.345} C_VEL
LIN {X 0,Y 320.551,Z 600.149,A -85,B 0,C 180,E1 -15196.045,E2 -15196.045} C_VEL
LIN {X 0,Y 319.405,Z 607.592,A -85,B 0,C 180,E1 -15197.935,E2 -15197.935} C_VEL
LIN {X 0,Y 318.663,Z 613.578,A -85,B 0,C 180,E1 -15199.838,E2 -15199.838} C_VEL
LIN {X 0,Y 318.194,Z 618.313,A -85,B 0,C 180,E1 -15201.746,E2 -15201.746} C_VEL
LIN {X 0,Y 317.908,Z 621.933,A -85,B 0,C 180,E1 -15203.654,E2 -15203.654} C_VEL
LIN {X 0,Y 317.81,Z 623.801,A -85,B 0,C 180,E1 -15204.925,E2 -15204.925} C_VEL
LIN {X 0,Y 317.81,Z 625.204,A -85,B 0,C 180,E1 -15206.196,E2 -15206.196} C_VEL
LIN {X 0,Y 317.78,Z 626.204,A -85,B 0,C 180,E1 -15207.465,E2 -15207.465} C_VEL
LIN {X 0,Y 317.799,Z 626.815,A -85,B 0,C 180,E1 -15208.733,E2 -15208.733} C_VEL
LIN {X 0,Y 317.852,Z 627.032,A -85,B 0,C 180,E1 -15210,E2 -15210} C_VEL
LIN {X 0,Y 317.799,Z 626.809,A -85,B 0,C 180,E1 -15211.267,E2 -15211.267} C_VEL
LIN {X 0,Y 317.78,Z 626.195,A -85,B 0,C 180,E1 -15212.535,E2 -15212.535} C_VEL
LIN {X 0,Y 317.809,Z 625.191,A -85,B 0,C 180,E1 -15213.804,E2 -15213.804} C_VEL
LIN {X 0,Y 317.838,Z 622.883,A -85,B 0,C 180,E1 -15215.711,E2 -15215.711} C_VEL
LIN {X 0,Y 318.067,Z 619.593,A -85,B 0,C 180,E1 -15217.618,E2 -15217.618} C_VEL
LIN {X 0,Y 318.48,Z 615.231,A -85,B 0,C 180,E1 -15219.526,E2 -15219.526} C_VEL
LIN {X 0,Y 319.091,Z 609.678,A -85,B 0,C 180,E1 -15221.433,E2 -15221.433} C_VEL
LIN {X 0,Y 320.119,Z 602.759,A -85,B 0,C 180,E1 -15223.327,E2 -15223.327} C_VEL
LIN {X 0,Y 321.134,Z 595.695,A -85,B 0,C 180,E1 -15224.901,E2 -15224.901} C_VEL
LIN {X 0,Y 322.33,Z 587.184,A -85,B 0,C 180,E1 -15226.466,E2 -15226.466} C_VEL
LIN {X 0,Y 323.74,Z 576.672,A -85,B 0,C 180,E1 -15228.02,E2 -15228.02} C_VEL
LIN {X 0,Y 325.372,Z 564.85,A -85,B 0,C 180,E1 -15229.396,E2 -15229.396} C_VEL
LIN {X 0,Y 326.72,Z 552.949,A -85,B 0,C 180,E1 -15230.459,E2 -15230.459} C_VEL
LIN {X 0,Y 327.916,Z 540.568,A -85,B 0,C 180,E1 -15231.285,E2 -15231.285} C_VEL
LIN {X 0,Y 328.843,Z 527.835,A -85,B 0,C 180,E1 -15231.88,E2 -15231.88} C_VEL
LIN {X 0,Y 329.391,Z 514.417,A -85,B 0,C 180,E1 -15232.254,E2 -15232.254} C_VEL
LIN {X 0,Y 330.601,Z 454.95,A -85,B 0,C 180,E1 -15233.54,E2 -15233.54} C_VEL
LIN {X 0,Y 326.336,Z 427.57,A -85,B 0,C 180,E1 -15234.507,E2 -15234.507} C_VEL
LIN {X 0,Y 323.908,Z 414.05,A -85,B 0,C 180,E1 -15235.056,E2 -15235.056} C_VEL
LIN {X 0,Y 324.38,Z 410.349,A -85,B 0,C 180,E1 -15236.023,E2 -15236.023} C_VEL
LIN {X 0,Y 323.162,Z 402.642,A -85,B 0,C 180,E1 -15238.229,E2 -15238.229} C_VEL
LIN {X 0,Y 320.89,Z 392.322,A -85,B 0,C 180,E1 -15241.332,E2 -15241.332} C_VEL
LIN {X 0,Y 319.57,Z 386.682,A -85,B 0,C 180,E1 -15243.137,E2 -15243.137} C_VEL
LIN {X 0,Y 319.558,Z 386.679,A -85,B 0,C 180,E1 -15246.427,E2 -15246.427} C_VEL
LIN {X 0,Y 319.558,Z 386.682,A -85,B 0,C 180,E1 -15249.668,E2 -15249.668} C_VEL
LIN {X 0,Y 319.562,Z 386.68,A -85,B 0,C 180,E1 -15253.468,E2 -15253.468} C_VEL
LIN {X 0,Y 319.601,Z 386.671,A -85,B 0,C 180,E1 -15257.024,E2 -15257.024} C_VEL
LIN {X 0,Y 319.581,Z 386.674,A -85,B 0,C 180,E1 -15260.376,E2 -15260.376} C_VEL
LIN {X 0,Y 319.555,Z 386.681,A -85,B 0,C 180,E1 -15263.572,E2 -15263.572} C_VEL
LIN {X 0,Y 319.572,Z 386.674,A -85,B 0,C 180,E1 -15266.686,E2 -15266.686} C_VEL
LIN {X 0,Y 319.586,Z 386.675,A -85,B 0,C 180,E1 -15269.616,E2 -15269.616} C_VEL
LIN {X 0,Y 319.603,Z 386.669,A -85,B 0,C 180,E1 -15272.498,E2 -15272.498} C_VEL
LIN {X 0,Y 319.599,Z 386.674,A -85,B 0,C 180,E1 -15275.304,E2 -15275.304} C_VEL
LIN {X 0,Y 319.591,Z 386.671,A -85,B 0,C 180,E1 -15278.047,E2 -15278.047} C_VEL
LIN {X 0,Y 319.683,Z 386.664,A -85,B 0,C 180,E1 -15280.962,E2 -15280.962} C_VEL
LIN {X 0,Y 319.724,Z 386.66,A -85,B 0,C 180,E1 -15285.276,E2 -15285.276} C_VEL
LIN {X 0,Y 319.753,Z 386.648,A -85,B 0,C 180,E1 -15289.873,E2 -15289.873} C_VEL
LIN {X 0,Y 319.926,Z 386.631,A -85,B 0,C 180,E1 -15292.426,E2 -15292.426} C_VEL
LIN {X 0,Y 319.742,Z 386.657,A -85,B 0,C 180,E1 -15294.956,E2 -15294.956} C_VEL
LIN {X 0,Y 319.985,Z 386.621,A -85,B 0,C 180,E1 -15297.482,E2 -15297.482} C_VEL
LIN {X 0,Y 320.162,Z 386.601,A -85,B 0,C 180,E1 -15300,E2 -15300} C_VEL
LIN {X 0,Y 319.985,Z 386.625,A -85,B 0,C 180,E1 -15302.518,E2 -15302.518} C_VEL
LIN {X 0,Y 319.924,Z 386.628,A -85,B 0,C 180,E1 -15306.675,E2 -15306.675} C_VEL
LIN {X 0,Y 319.753,Z 386.652,A -85,B 0,C 180,E1 -15310.127,E2 -15310.127} C_VEL
LIN {X 0,Y 319.725,Z 386.66,A -85,B 0,C 180,E1 -15314.724,E2 -15314.724} C_VEL
LIN {X 0,Y 319.683,Z 386.659,A -85,B 0,C 180,E1 -15319.038,E2 -15319.038} C_VEL
LIN {X 0,Y 319.564,Z 386.676,A -85,B 0,C 180,E1 -15323.32,E2 -15323.32} C_VEL
LIN {X 0,Y 319.629,Z 386.666,A -85,B 0,C 180,E1 -15326.089,E2 -15326.089} C_VEL
LIN {X 0,Y 319.584,Z 386.676,A -85,B 0,C 180,E1 -15328.934,E2 -15328.934} C_VEL
LIN {X 0,Y 319.527,Z 386.678,A -85,B 0,C 180,E1 -15331.863,E2 -15331.863} C_VEL
LIN {X 0,Y 319.575,Z 386.674,A -85,B 0,C 180,E1 -15335.544,E2 -15335.544} C_VEL
LIN {X 0,Y 319.596,Z 386.673,A -85,B 0,C 180,E1 -15338.005,E2 -15338.005} C_VEL
LIN {X 0,Y 319.594,Z 386.671,A -85,B 0,C 180,E1 -15341.612,E2 -15341.612} C_VEL
LIN {X 0,Y 319.54,Z 386.678,A -85,B 0,C 180,E1 -15345.268,E2 -15345.268} C_VEL
LIN {X 0,Y 319.527,Z 386.683,A -85,B 0,C 180,E1 -15348.713,E2 -15348.713} C_VEL
LIN {X 0,Y 319.577,Z 386.68,A -85,B 0,C 180,E1 -15352.345,E2 -15352.345} C_VEL
LIN {X 0,Y 319.56,Z 386.678,A -85,B 0,C 180,E1 -15355.124,E2 -15355.124} C_VEL
LIN {X 0,Y 319.566,Z 386.677,A -85,B 0,C 180,E1 -15359.06,E2 -15359.06} C_VEL
LIN {X 0,Y 319.688,Z 386.742,A -85,B 0,C 180,E1 -15362.639,E2 -15362.639} C_VEL
LIN {X 0,Y 321.052,Z 393.126,A -85,B 0,C 180,E1 -15364.809,E2 -15364.809} C_VEL
LIN {X 0,Y 329.893,Z 415.63,A -85,B 0,C 180,E1 -15366.066,E2 -15366.066} C_VEL
LIN {X 0,Y 331.303,Z 423.006,A -85,B 0,C 180,E1 -15366.347,E2 -15366.347} C_VEL
LIN {X 0,Y 329.536,Z 500.266,A -85,B 0,C 180,E1 -15368.045,E2 -15368.045} C_VEL
LIN {X 0,Y 328.782,Z 513.26,A -85,B 0,C 180,E1 -15368.569,E2 -15368.569} C_VEL
LIN {X 0,Y 327.979,Z 525.254,A -85,B 0,C 180,E1 -15369.295,E2 -15369.295} C_VEL
LIN {X 0,Y 326.903,Z 536.578,A -85,B 0,C 180,E1 -15370.209,E2 -15370.209} C_VEL
LIN {X 0,Y 325.525,Z 548.471,A -85,B 0,C 180,E1 -15371.464,E2 -15371.464} C_VEL
LIN {X 0,Y 324.38,Z 558.689,A -85,B 0,C 180,E1 -15372.837,E2 -15372.837} C_VEL
LIN {X 0,Y 323.092,Z 567.182,A -85,B 0,C 180,E1 -15374.223,E2 -15374.223} C_VEL
LIN {X 0,Y 321.869,Z 575.04,A -85,B 0,C 180,E1 -15375.781,E2 -15375.781} C_VEL
LIN {X 0,Y 320.665,Z 582.716,A -85,B 0,C 180,E1 -15377.662,E2 -15377.662} C_VEL
LIN {X 0,Y 319.577,Z 589.758,A -85,B 0,C 180,E1 -15379.867,E2 -15379.867} C_VEL
LIN {X 0,Y 318.862,Z 594.447,A -85,B 0,C 180,E1 -15381.763,E2 -15381.763} C_VEL
LIN {X 0,Y 318.468,Z 598.03,A -85,B 0,C 180,E1 -15383.665,E2 -15383.665} C_VEL
LIN {X 0,Y 318.254,Z 599.882,A -85,B 0,C 180,E1 -15384.932,E2 -15384.932} C_VEL
LIN {X 0,Y 318.051,Z 601.277,A -85,B 0,C 180,E1 -15386.199,E2 -15386.199} C_VEL
LIN {X 0,Y 317.858,Z 602.879,A -85,B 0,C 180,E1 -15388.733,E2 -15388.733} C_VEL
LIN {X 0,Y 317.859,Z 603.109,A -85,B 0,C 180,E1 -15390,E2 -15390} C_VEL
LIN {X 0,Y 317.858,Z 602.919,A -85,B 0,C 180,E1 -15391.267,E2 -15391.267} C_VEL
LIN {X 0,Y 318.049,Z 601.369,A -85,B 0,C 180,E1 -15393.801,E2 -15393.801} C_VEL
LIN {X 0,Y 318.253,Z 600.015,A -85,B 0,C 180,E1 -15395.068,E2 -15395.068} C_VEL
LIN {X 0,Y 318.629,Z 597.119,A -85,B 0,C 180,E1 -15396.989,E2 -15396.989} C_VEL
LIN {X 0,Y 319.052,Z 593.278,A -85,B 0,C 180,E1 -15398.87,E2 -15398.87} C_VEL
LIN {X 0,Y 319.813,Z 588.27,A -85,B 0,C 180,E1 -15400.765,E2 -15400.765} C_VEL
LIN {X 0,Y 320.784,Z 581.964,A -85,B 0,C 180,E1 -15402.655,E2 -15402.655} C_VEL
LIN {X 0,Y 322.005,Z 574.067,A -85,B 0,C 180,E1 -15404.536,E2 -15404.536} C_VEL
LIN {X 0,Y 323.314,Z 566.01,A -85,B 0,C 180,E1 -15406.09,E2 -15406.09} C_VEL
LIN {X 0,Y 324.612,Z 556.183,A -85,B 0,C 180,E1 -15407.644,E2 -15407.644} C_VEL
LIN {X 0,Y 325.751,Z 546.51,A -85,B 0,C 180,E1 -15408.882,E2 -15408.882} C_VEL
LIN {X 0,Y 326.998,Z 536.027,A -85,B 0,C 180,E1 -15409.949,E2 -15409.949} C_VEL
LIN {X 0,Y 328.218,Z 523.398,A -85,B 0,C 180,E1 -15410.935,E2 -15410.935} C_VEL
LIN {X 0,Y 329.022,Z 510.751,A -85,B 0,C 180,E1 -15411.662,E2 -15411.662} C_VEL
LIN {X 0,Y 329.66,Z 498.695,A -85,B 0,C 180,E1 -15412.111,E2 -15412.111} C_VEL
LIN {X 0,Y 331.237,Z 421.981,A -85,B 0,C 180,E1 -15413.793,E2 -15413.793} C_VEL
LIN {X 0,Y 329.469,Z 414.44,A -85,B 0,C 180,E1 -15414.107,E2 -15414.107} C_VEL
LIN {X 0,Y 321.758,Z 395.056,A -85,B 0,C 180,E1 -15415.198,E2 -15415.198} C_VEL
LIN {X 0,Y 321.008,Z 392.89,A -85,B 0,C 180,E1 -15415.333,E2 -15415.333} C_VEL
LIN {X 0,Y 319.65,Z 386.669,A -85,B 0,C 180,E1 -15417.569,E2 -15417.569} C_VEL
LIN {X 0,Y 319.566,Z 386.675,A -85,B 0,C 180,E1 -15420.94,E2 -15420.94} C_VEL
LIN {X 0,Y 319.559,Z 386.678,A -85,B 0,C 180,E1 -15424.876,E2 -15424.876} C_VEL
LIN {X 0,Y 319.559,Z 386.679,A -85,B 0,C 180,E1 -15427.37,E2 -15427.37} C_VEL
LIN {X 0,Y 318.927,Z 386.762,A -85,B 0,C 180,E1 -15428.422,E2 -15428.422} C_VEL
LIN {X 0,Y 316.067,Z 387.117,A -85,B 0,C 180,E1 -15430.133,E2 -15430.133} C_VEL
LIN {X 0,Y 313.616,Z 387.42,A -85,B 0,C 180,E1 -15431.52,E2 -15431.52} C_VEL
LIN {X 0,Y 312.56,Z 387.548,A -85,B 0,C 180,E1 -15432.595,E2 -15432.595} C_VEL
LIN {X 0,Y 312.474,Z 387.557,A -85,B 0,C 180,E1 -15432.959,E2 -15432.959} C_VEL
LIN {X 0,Y 312.534,Z 387.549,A -85,B 0,C 180,E1 -15436.019,E2 -15436.019} C_VEL
LIN {X 0,Y 312.527,Z 387.557,A -85,B 0,C 180,E1 -15439.868,E2 -15439.868} C_VEL
LIN {X 0,Y 312.549,Z 387.547,A -85,B 0,C 180,E1 -15442.618,E2 -15442.618} C_VEL
LIN {X 0,Y 312.515,Z 387.552,A -85,B 0,C 180,E1 -15446.31,E2 -15446.31} C_VEL
LIN {X 0,Y 312.54,Z 387.55,A -85,B 0,C 180,E1 -15450.349,E2 -15450.349} C_VEL
LIN {X 0,Y 312.597,Z 387.545,A -85,B 0,C 180,E1 -15454.064,E2 -15454.064} C_VEL
LIN {X 0,Y 312.582,Z 387.548,A -85,B 0,C 180,E1 -15457.528,E2 -15457.528} C_VEL
LIN {X 0,Y 312.632,Z 387.539,A -85,B 0,C 180,E1 -15461.656,E2 -15461.656} C_VEL
LIN {X 0,Y 312.688,Z 387.535,A -85,B 0,C 180,E1 -15465.686,E2 -15465.686} C_VEL
LIN {X 0,Y 312.697,Z 387.532,A -85,B 0,C 180,E1 -15469.642,E2 -15469.642} C_VEL
LIN {X 0,Y 312.865,Z 387.511,A -85,B 0,C 180,E1 -15472.254,E2 -15472.254} C_VEL
LIN {X 0,Y 312.712,Z 387.53,A -85,B 0,C 180,E1 -15474.842,E2 -15474.842} C_VEL
LIN {X 0,Y 312.986,Z 387.497,A -85,B 0,C 180,E1 -15478.713,E2 -15478.713} C_VEL
LIN {X 0,Y 313.114,Z 387.479,A -85,B 0,C 180,E1 -15480,E2 -15480} C_VEL
LIN {X 0,Y 312.932,Z 387.498,A -85,B 0,C 180,E1 -15482.574,E2 -15482.574} C_VEL
LIN {X 0,Y 312.903,Z 387.506,A -85,B 0,C 180,E1 -15486.448,E2 -15486.448} C_VEL
LIN {X 0,Y 312.781,Z 387.522,A -85,B 0,C 180,E1 -15489.049,E2 -15489.049} C_VEL
LIN {X 0,Y 312.631,Z 387.541,A -85,B 0,C 180,E1 -15492.991,E2 -15492.991} C_VEL
LIN {X 0,Y 312.632,Z 387.539,A -85,B 0,C 180,E1 -15495.65,E2 -15495.65} C_VEL
LIN {X 0,Y 312.624,Z 387.539,A -85,B 0,C 180,E1 -15499.237,E2 -15499.237} C_VEL
LIN {X 0,Y 312.54,Z 387.556,A -85,B 0,C 180,E1 -15502.79,E2 -15502.79} C_VEL
LIN {X 0,Y 312.577,Z 387.551,A -85,B 0,C 180,E1 -15506.723,E2 -15506.723} C_VEL
LIN {X 0,Y 312.54,Z 387.551,A -85,B 0,C 180,E1 -15509.651,E2 -15509.651} C_VEL
LIN {X 0,Y 312.515,Z 387.551,A -85,B 0,C 180,E1 -15513.689,E2 -15513.689} C_VEL
LIN {X 0,Y 312.537,Z 387.549,A -85,B 0,C 180,E1 -15517.384,E2 -15517.384} C_VEL
LIN {X 0,Y 312.522,Z 387.555,A -85,B 0,C 180,E1 -15520.704,E2 -15520.704} C_VEL
LIN {X 0,Y 312.53,Z 387.553,A -85,B 0,C 180,E1 -15524.196,E2 -15524.196} C_VEL
LIN {X 0,Y 312.516,Z 387.556,A -85,B 0,C 180,E1 -15527.912,E2 -15527.912} C_VEL
LIN {X 0,Y 312.535,Z 387.555,A -85,B 0,C 180,E1 -15531.911,E2 -15531.911} C_VEL
LIN {X 0,Y 312.505,Z 387.56,A -85,B 0,C 180,E1 -15535.791,E2 -15535.791} C_VEL
LIN {X 0,Y 312.551,Z 387.742,A -85,B 0,C 180,E1 -15536.43,E2 -15536.43} C_VEL
LIN {X 0,Y 315.029,Z 398.434,A -85,B 0,C 180,E1 -15539.832,E2 -15539.832} C_VEL
LIN {X 0,Y 317.192,Z 409.138,A -85,B 0,C 180,E1 -15543.06,E2 -15543.06} C_VEL
LIN {X 0,Y 317.468,Z 411.418,A -85,B 0,C 180,E1 -15543.721,E2 -15543.721} C_VEL
LIN {X 0,Y 317.26,Z 413.845,A -85,B 0,C 180,E1 -15544.38,E2 -15544.38} C_VEL
LIN {X 0,Y 322.959,Z 447.398,A -85,B 0,C 180,E1 -15545.674,E2 -15545.674} C_VEL
LIN {X 0,Y 324.106,Z 457.168,A -85,B 0,C 180,E1 -15545.996,E2 -15545.996} C_VEL
LIN {X 0,Y 322.606,Z 522.526,A -85,B 0,C 180,E1 -15547.464,E2 -15547.464} C_VEL
LIN {X 0,Y 321.719,Z 535.705,A -85,B 0,C 180,E1 -15547.99,E2 -15547.99} C_VEL
LIN {X 0,Y 320.609,Z 547.821,A -85,B 0,C 180,E1 -15548.712,E2 -15548.712} C_VEL
LIN {X 0,Y 319.242,Z 560.056,A -85,B 0,C 180,E1 -15549.713,E2 -15549.713} C_VEL
LIN {X 0,Y 317.713,Z 571.642,A -85,B 0,C 180,E1 -15550.957,E2 -15550.957} C_VEL
LIN {X 0,Y 316.129,Z 582.076,A -85,B 0,C 180,E1 -15552.368,E2 -15552.368} C_VEL
LIN {X 0,Y 314.963,Z 590.71,A -85,B 0,C 180,E1 -15553.822,E2 -15553.822} C_VEL
LIN {X 0,Y 313.625,Z 599.882,A -85,B 0,C 180,E1 -15555.73,E2 -15555.73} C_VEL
LIN {X 0,Y 312.41,Z 607.324,A -85,B 0,C 180,E1 -15557.66,E2 -15557.66} C_VEL
LIN {X 0,Y 311.642,Z 613.311,A -85,B 0,C 180,E1 -15559.606,E2 -15559.606} C_VEL
LIN {X 0,Y 311.137,Z 618.046,A -85,B 0,C 180,E1 -15561.557,E2 -15561.557} C_VEL
LIN {X 0,Y 310.831,Z 621.666,A -85,B 0,C 180,E1 -15563.509,E2 -15563.509} C_VEL
LIN {X 0,Y 310.714,Z 623.533,A -85,B 0,C 180,E1 -15564.809,E2 -15564.809} C_VEL
LIN {X 0,Y 310.72,Z 624.937,A -85,B 0,C 180,E1 -15566.109,E2 -15566.109} C_VEL
LIN {X 0,Y 310.702,Z 625.938,A -85,B 0,C 180,E1 -15567.407,E2 -15567.407} C_VEL
LIN {X 0,Y 310.71,Z 626.549,A -85,B 0,C 180,E1 -15568.704,E2 -15568.704} C_VEL
LIN {X 0,Y 310.759,Z 626.765,A -85,B 0,C 180,E1 -15570,E2 -15570} C_VEL
LIN {X 0,Y 310.71,Z 626.542,A -85,B 0,C 180,E1 -15571.296,E2 -15571.296} C_VEL
LIN {X 0,Y 310.702,Z 625.928,A -85,B 0,C 180,E1 -15572.593,E2 -15572.593} C_VEL
LIN {X 0,Y 310.719,Z 624.924,A -85,B 0,C 180,E1 -15573.891,E2 -15573.891} C_VEL
LIN {X 0,Y 310.766,Z 622.821,A -85,B 0,C 180,E1 -15575.694,E2 -15575.694} C_VEL
LIN {X 0,Y 311.009,Z 619.324,A -85,B 0,C 180,E1 -15577.792,E2 -15577.792} C_VEL
LIN {X 0,Y 311.431,Z 614.961,A -85,B 0,C 180,E1 -15579.744,E2 -15579.744} C_VEL
LIN {X 0,Y 312.092,Z 609.408,A -85,B 0,C 180,E1 -15581.693,E2 -15581.693} C_VEL
LIN {X 0,Y 313.194,Z 602.489,A -85,B 0,C 180,E1 -15583.628,E2 -15583.628} C_VEL
LIN {X 0,Y 314.541,Z 593.833,A -85,B 0,C 180,E1 -15585.552,E2 -15585.552} C_VEL
LIN {X 0,Y 315.765,Z 584.957,A -85,B 0,C 180,E1 -15587.151,E2 -15587.151} C_VEL
LIN {X 0,Y 317.17,Z 575.224,A -85,B 0,C 180,E1 -15588.573,E2 -15588.573} C_VEL
LIN {X 0,Y 318.674,Z 564.578,A -85,B 0,C 180,E1 -15589.82,E2 -15589.82} C_VEL
LIN {X 0,Y 320.066,Z 552.676,A -85,B 0,C 180,E1 -15590.904,E2 -15590.904} C_VEL
LIN {X 0,Y 321.285,Z 540.293,A -85,B 0,C 180,E1 -15591.746,E2 -15591.746} C_VEL
LIN {X 0,Y 322.274,Z 527.557,A -85,B 0,C 180,E1 -15592.35,E2 -15592.35} C_VEL
LIN {X 0,Y 322.847,Z 514.13,A -85,B 0,C 180,E1 -15592.73,E2 -15592.73} C_VEL
LIN {X 0,Y 323.963,Z 454.953,A -85,B 0,C 180,E1 -15594.045,E2 -15594.045} C_VEL
LIN {X 0,Y 319.273,Z 425.036,A -85,B 0,C 180,E1 -15595.14,E2 -15595.14} C_VEL
LIN {X 0,Y 317.204,Z 413.835,A -85,B 0,C 180,E1 -15595.607,E2 -15595.607} C_VEL
LIN {X 0,Y 317.355,Z 410.208,A -85,B 0,C 180,E1 -15596.604,E2 -15596.604} C_VEL
LIN {X 0,Y 315.398,Z 400.006,A -85,B 0,C 180,E1 -15599.653,E2 -15599.653} C_VEL
LIN {X 0,Y 312.511,Z 387.562,A -85,B 0,C 180,E1 -15603.618,E2 -15603.618} C_VEL
LIN {X 0,Y 312.537,Z 387.553,A -85,B 0,C 180,E1 -15607.383,E2 -15607.383} C_VEL
LIN {X 0,Y 312.491,Z 387.558,A -85,B 0,C 180,E1 -15610.708,E2 -15610.708} C_VEL
LIN {X 0,Y 312.507,Z 387.552,A -85,B 0,C 180,E1 -15614.198,E2 -15614.198} C_VEL
LIN {X 0,Y 312.545,Z 387.552,A -85,B 0,C 180,E1 -15617.905,E2 -15617.905} C_VEL
LIN {X 0,Y 312.541,Z 387.552,A -85,B 0,C 180,E1 -15621.907,E2 -15621.907} C_VEL
LIN {X 0,Y 312.502,Z 387.556,A -85,B 0,C 180,E1 -15625.789,E2 -15625.789} C_VEL
LIN {X 0,Y 312.518,Z 387.555,A -85,B 0,C 180,E1 -15628.853,E2 -15628.853} C_VEL
LIN {X 0,Y 312.569,Z 387.546,A -85,B 0,C 180,E1 -15631.824,E2 -15631.824} C_VEL
LIN {X 0,Y 312.58,Z 387.546,A -85,B 0,C 180,E1 -15634.71,E2 -15634.71} C_VEL
LIN {X 0,Y 312.581,Z 387.547,A -85,B 0,C 180,E1 -15637.528,E2 -15637.528} C_VEL
LIN {X 0,Y 312.632,Z 387.538,A -85,B 0,C 180,E1 -15641.656,E2 -15641.656} C_VEL
LIN {X 0,Y 312.688,Z 387.534,A -85,B 0,C 180,E1 -15645.686,E2 -15645.686} C_VEL
LIN {X 0,Y 312.697,Z 387.527,A -85,B 0,C 180,E1 -15649.642,E2 -15649.642} C_VEL
LIN {X 0,Y 312.865,Z 387.51,A -85,B 0,C 180,E1 -15652.254,E2 -15652.254} C_VEL
LIN {X 0,Y 312.713,Z 387.533,A -85,B 0,C 180,E1 -15654.842,E2 -15654.842} C_VEL
LIN {X 0,Y 312.986,Z 387.495,A -85,B 0,C 180,E1 -15658.713,E2 -15658.713} C_VEL
LIN {X 0,Y 313.114,Z 387.479,A -85,B 0,C 180,E1 -15660,E2 -15660} C_VEL
LIN {X 0,Y 312.932,Z 387.504,A -85,B 0,C 180,E1 -15662.575,E2 -15662.575} C_VEL
LIN {X 0,Y 312.886,Z 387.505,A -85,B 0,C 180,E1 -15666.658,E2 -15666.658} C_VEL
LIN {X 0,Y 312.782,Z 387.524,A -85,B 0,C 180,E1 -15669.049,E2 -15669.049} C_VEL
LIN {X 0,Y 312.631,Z 387.54,A -85,B 0,C 180,E1 -15672.991,E2 -15672.991} C_VEL
LIN {X 0,Y 312.632,Z 387.54,A -85,B 0,C 180,E1 -15675.65,E2 -15675.65} C_VEL
LIN {X 0,Y 312.625,Z 387.536,A -85,B 0,C 180,E1 -15679.237,E2 -15679.237} C_VEL
LIN {X 0,Y 312.54,Z 387.555,A -85,B 0,C 180,E1 -15682.79,E2 -15682.79} C_VEL
LIN {X 0,Y 312.597,Z 387.541,A -85,B 0,C 180,E1 -15685.936,E2 -15685.936} C_VEL
LIN {X 0,Y 312.54,Z 387.551,A -85,B 0,C 180,E1 -15689.651,E2 -15689.651} C_VEL
LIN {X 0,Y 312.515,Z 387.554,A -85,B 0,C 180,E1 -15693.69,E2 -15693.69} C_VEL
LIN {X 0,Y 312.549,Z 387.548,A -85,B 0,C 180,E1 -15697.382,E2 -15697.382} C_VEL
LIN {X 0,Y 312.523,Z 387.554,A -85,B 0,C 180,E1 -15700.704,E2 -15700.704} C_VEL
LIN {X 0,Y 312.53,Z 387.556,A -85,B 0,C 180,E1 -15704.196,E2 -15704.196} C_VEL
LIN {X 0,Y 312.485,Z 387.56,A -85,B 0,C 180,E1 -15707.919,E2 -15707.919} C_VEL
LIN {X 0,Y 312.534,Z 387.555,A -85,B 0,C 180,E1 -15711.911,E2 -15711.911} C_VEL
LIN {X 0,Y 312.506,Z 387.559,A -85,B 0,C 180,E1 -15715.791,E2 -15715.791} C_VEL
LIN {X 0,Y 312.52,Z 387.556,A -85,B 0,C 180,E1 -15718.854,E2 -15718.854} C_VEL
LIN {X 0,Y 312.615,Z 387.674,A -85,B 0,C 180,E1 -15722.194,E2 -15722.194} C_VEL
LIN {X 0,Y 313.817,Z 393.172,A -85,B 0,C 180,E1 -15724.165,E2 -15724.165} C_VEL
LIN {X 0,Y 323.539,Z 417.416,A -85,B 0,C 180,E1 -15725.601,E2 -15725.601} C_VEL
LIN {X 0,Y 324.814,Z 423.609,A -85,B 0,C 180,E1 -15725.852,E2 -15725.852} C_VEL
LIN {X 0,Y 323.027,Z 499.391,A -85,B 0,C 180,E1 -15727.537,E2 -15727.537} C_VEL
LIN {X 0,Y 322.242,Z 512.778,A -85,B 0,C 180,E1 -15728.07,E2 -15728.07} C_VEL
LIN {X 0,Y 321.354,Z 525.529,A -85,B 0,C 180,E1 -15728.848,E2 -15728.848} C_VEL
LIN {X 0,Y 320.249,Z 536.851,A -85,B 0,C 180,E1 -15729.78,E2 -15729.78} C_VEL
LIN {X 0,Y 318.803,Z 548.743,A -85,B 0,C 180,E1 -15731.058,E2 -15731.058} C_VEL
LIN {X 0,Y 317.59,Z 559.128,A -85,B 0,C 180,E1 -15732.485,E2 -15732.485} C_VEL
LIN {X 0,Y 316.276,Z 567.452,A -85,B 0,C 180,E1 -15733.874,E2 -15733.874} C_VEL
LIN {X 0,Y 314.998,Z 575.309,A -85,B 0,C 180,E1 -15735.464,E2 -15735.464} C_VEL
LIN {X 0,Y 313.739,Z 582.984,A -85,B 0,C 180,E1 -15737.385,E2 -15737.385} C_VEL
LIN {X 0,Y 312.577,Z 590.027,A -85,B 0,C 180,E1 -15739.638,E2 -15739.638} C_VEL
LIN {X 0,Y 311.838,Z 594.716,A -85,B 0,C 180,E1 -15741.576,E2 -15741.576} C_VEL
LIN {X 0,Y 311.402,Z 598.299,A -85,B 0,C 180,E1 -15743.521,E2 -15743.521} C_VEL
LIN {X 0,Y 311.185,Z 600.15,A -85,B 0,C 180,E1 -15744.817,E2 -15744.817} C_VEL
LIN {X 0,Y 310.987,Z 601.544,A -85,B 0,C 180,E1 -15746.113,E2 -15746.113} C_VEL
LIN {X 0,Y 310.769,Z 603.146,A -85,B 0,C 180,E1 -15748.704,E2 -15748.704} C_VEL
LIN {X 0,Y 310.767,Z 603.376,A -85,B 0,C 180,E1 -15750,E2 -15750} C_VEL
LIN {X 0,Y 310.768,Z 603.186,A -85,B 0,C 180,E1 -15751.296,E2 -15751.296} C_VEL
LIN {X 0,Y 310.986,Z 601.635,A -85,B 0,C 180,E1 -15753.887,E2 -15753.887} C_VEL
LIN {X 0,Y 311.184,Z 600.281,A -85,B 0,C 180,E1 -15755.183,E2 -15755.183} C_VEL
LIN {X 0,Y 311.553,Z 597.632,A -85,B 0,C 180,E1 -15756.996,E2 -15756.996} C_VEL
LIN {X 0,Y 312.026,Z 593.545,A -85,B 0,C 180,E1 -15759.071,E2 -15759.071} C_VEL
LIN {X 0,Y 312.846,Z 588.536,A -85,B 0,C 180,E1 -15761.008,E2 -15761.008} C_VEL
LIN {X 0,Y 313.871,Z 582.228,A -85,B 0,C 180,E1 -15762.939,E2 -15762.939} C_VEL
LIN {X 0,Y 315.123,Z 574.332,A -85,B 0,C 180,E1 -15764.861,E2 -15764.861} C_VEL
LIN {X 0,Y 316.493,Z 566.275,A -85,B 0,C 180,E1 -15766.446,E2 -15766.446} C_VEL
LIN {X 0,Y 317.874,Z 556.232,A -85,B 0,C 180,E1 -15768.064,E2 -15768.064} C_VEL
LIN {X 0,Y 319.224,Z 545.384,A -85,B 0,C 180,E1 -15769.45,E2 -15769.45} C_VEL
LIN {X 0,Y 320.507,Z 534.529,A -85,B 0,C 180,E1 -15770.538,E2 -15770.538} C_VEL
LIN {X 0,Y 321.698,Z 522.531,A -85,B 0,C 180,E1 -15771.464,E2 -15771.464} C_VEL
LIN {X 0,Y 322.511,Z 510.211,A -85,B 0,C 180,E1 -15772.164,E2 -15772.164} C_VEL
LIN {X 0,Y 323.165,Z 497.448,A -85,B 0,C 180,E1 -15772.622,E2 -15772.622} C_VEL
LIN {X 0,Y 324.768,Z 423.069,A -85,B 0,C 180,E1 -15774.277,E2 -15774.277} C_VEL
LIN {X 0,Y 323.31,Z 416.979,A -85,B 0,C 180,E1 -15774.541,E2 -15774.541} C_VEL
LIN {X 0,Y 315.47,Z 397.229,A -85,B 0,C 180,E1 -15775.689,E2 -15775.689} C_VEL
LIN {X 0,Y 313.829,Z 393.167,A -85,B 0,C 180,E1 -15775.957,E2 -15775.957} C_VEL
LIN {X 0,Y 312.581,Z 387.551,A -85,B 0,C 180,E1 -15777.991,E2 -15777.991} C_VEL
LIN {X 0,Y 312.514,Z 387.554,A -85,B 0,C 180,E1 -15781.288,E2 -15781.288} C_VEL
LIN {X 0,Y 312.506,Z 387.558,A -85,B 0,C 180,E1 -15784.209,E2 -15784.209} C_VEL
LIN {X 0,Y 312.533,Z 387.555,A -85,B 0,C 180,E1 -15788.089,E2 -15788.089} C_VEL
LIN {X 0,Y 312.485,Z 387.56,A -85,B 0,C 180,E1 -15792.081,E2 -15792.081} C_VEL
LIN {X 0,Y 312.474,Z 387.557,A -85,B 0,C 180,E1 -15792.959,E2 -15792.959} C_VEL
